// TwinCAT 3 PLC project VekSi_PLC
// ProgramVersion: 3.1.4026.22
// libraries:
//   Tc2_MC2, * (Beckhoff Automation GmbH)
//   Tc2_Standard, * (Beckhoff Automation GmbH)
//   Tc2_System, * (Beckhoff Automation GmbH)
//   Tc2_Utilities, * (Beckhoff Automation GmbH)
//   Tc3_IotBase, * (Beckhoff Automation GmbH)
//   Tc3_JsonXml, * (Beckhoff Automation GmbH)
// project tree:
//   Functions/ FB_CSVLogger.TcPOU, FB_ValveControl.TcPOU, FB_MqttManager.TcPOU, FB_SensorIO.TcPOU, MAIN.TcPOU
//   / PlcTask.TcTTO (not stored)
//   State_Var/ E_CSVLogState.TcDUT (not stored), E_MQTTState.TcDUT, E_CommandSource.TcDUT, E_ValveState.TcDUT, ST_MqttConfig.TcDUT, ST_MQTT_Command.TcDUT, ST_SensorData.TcDUT, ST_ValveData.TcDUT
//   Variables_Lists/ GVL_Config.TcGVL, GVL_HMI.TcGVL, GVL_IO.TcGVL, GVL_System.TcGVL
// real-time tasks:
//   TASK PlcTask: cycle T#10ms, priority 20, ADS port 350
// motion (NC):
//   TASK NC-Task 1 SAF: cycle T#2ms, priority 4, ADS port 501
//   TASK NC-Task 1 SVB: cycle T#10ms, priority 8, ADS port 511
//   AXIS Axis 2 (id 2)
//     Dynamic: Acceleration=16.9085, Deceleration=16.9085, Jerk=53.5391
//     Velo: RefSearch=3, RefSync=3, SlowManual=2, FastManual=3, Fast=3, Maximum=6
//     OtherSettings: AllowMotionCmdToSlave=true
//     encoder EncType=1
//       EncPara: ScaleFactorNumerator=0.003048
//         Inc: RefSoftSyncMask=#x0000ffff, HomingSensorSource=1
//         TimeComp: TimeCompMode=1, EncDelayCycles=4
//     drive DrvType=24
//       Analog: VeloReferenz=6.096, TorqueSetpointScale=10, ScaleFactorActTorque=0.1
//       TimeComp: TaskDelayCycles=1
//     controller CtrType=1
//       CtrPara: PriorControlFactor=1
//         PosDiffControl: Enable=false
//         Observer: BandWidth=20
//   AXIS Axis 3 (id 3)
//     Dynamic: Acceleration=16.9085, Deceleration=16.9085, Jerk=53.5391
//     Velo: RefSearch=3, RefSync=3, SlowManual=2, FastManual=3, Maximum=6
//     OtherSettings: AllowMotionCmdToSlave=true
//     encoder EncType=1
//       EncPara: ScaleFactorNumerator=0.003048
//         Inc: RefSoftSyncMask=#x0000ffff
//         TimeComp: TimeCompMode=1, EncDelayCycles=4
//     drive DrvType=24
//       Analog: VeloReferenz=6.096, TorqueSetpointScale=10, ScaleFactorActTorque=0.1
//       TimeComp: TaskDelayCycles=1
//     controller CtrType=1
//       CtrPara: PriorControlFactor=1
//         PosDiffControl: Enable=false
//         Observer: BandWidth=20
//   AXIS Axis 1 (id 1)
//     Dynamic: Acceleration=16.9085, Deceleration=16.9085, Jerk=53.5391
//     Velo: RefSearch=3, RefSync=3, SlowManual=2, FastManual=3, Maximum=6
//     OtherSettings: AllowMotionCmdToSlave=true
//     encoder EncType=1
//       EncPara: ScaleFactorNumerator=0.003048
//         Inc: RefSearchInverse=true, RefSyncInverse=false, RefSoftSyncMask=#x0000ffff
//         TimeComp: TimeCompMode=1, EncDelayCycles=4
//     drive DrvType=24
//       Analog: VeloReferenz=6.096, TorqueSetpointScale=10, ScaleFactorActTorque=0.1
//       TimeComp: TaskDelayCycles=1
//     controller CtrType=1
//       CtrPara: PriorControlFactor=1
//         PosDiffControl: Enable=false
//         Observer: BandWidth=20
// I/O:
//   DEVICE Device 1 (EtherCAT), AmsNetId 10.1.176.203.2.1
//     Term 1 (EK1200) [EK1200-5000 EtherCAT Power supply (2A E-Bus)]
//       Term 2 (EL6070-0033) [EL6070-0033 1Ch. Licence key terminal, individual licences]
//       Term 3 (EL1859) [EL1859 8Ch. Dig. Input 24V, 3ms, 8Ch. Dig. Output 24V, 0.5A]
//       Term 4 (EL3202) [EL3202 2Ch. Ana. Input PT100 (RTD)]
//       Term 5 (EL1004) [EL1004 4Ch. Dig. Input 24V, 3ms]
//       Term 6 (EL3074) [EL3074 4Ch. Ana. Input +/-10V, +/-20mA]
//       Term 7 (EK1322) [EK1322 2-port EtherCAT P junction with feed-in]
//         Box 8 (EPP7041-1002) [EPP7041-1002 1Ch. Stepper motor output stage (50V, 1.5A)]
//       Term 9 (EK1521-0010) [EK1521-0010 1 port EtherCAT junction (FX-SingleMode)]
//         Term 10 (EK1501-0010) [EK1501-0010 EtherCAT Coupler (2A E-Bus, FX-SingleMode, ID switch)]
//           Term 11 (EL3202) [EL3202 2Ch. Ana. Input PT100 (RTD)]
//           Term 12 (EL1859) [EL1859 8Ch. Dig. Input 24V, 3ms, 8Ch. Dig. Output 24V, 0.5A]
//           Term 13 (EL3074) [EL3074 4Ch. Ana. Input +/-10V, +/-20mA]
//           Term 22 (EL9011) [EL9011 End Terminal]
//       Term 14 (EK1521-0010) [EK1521-0010 1 port EtherCAT junction (FX-SingleMode)]
//         Term 15 (EK1501-0010) [EK1501-0010 EtherCAT Coupler (2A E-Bus, FX-SingleMode, ID switch)]
//           Term 16 (EL3202) [EL3202 2Ch. Ana. Input PT100 (RTD)]
//           Term 17 (EL1004) [EL1004 4Ch. Dig. Input 24V, 3ms]
//           Term 18 (EL3074) [EL3074 4Ch. Ana. Input +/-10V, +/-20mA]
//           Term 19 (EK1322) [EK1322 2-port EtherCAT P junction with feed-in]
//             Box 20 (EPP7041-1002) [EPP7041-1002 1Ch. Stepper motor output stage (50V, 1.5A)]
//             Box 21 (EPP7041-1002) [EPP7041-1002 1Ch. Stepper motor output stage (50V, 1.5A)]
// variable links:
//   NC-Task 1 SAF/Axes/Axis 1 <-> Device 1 (EtherCAT)/Term 1 (EK1200)/Term 7 (EK1322)/Box 8 (EPP7041-1002)
//     Drive/Inputs/In/nState1 @bit 3 <-> STM Status/Status/Error
//     Drive/Inputs/In/nState1 @bit 7 <-> STM Status/Status/Motor stall
//     Drive/Inputs/In/nState1 @bit 5 <-> STM Status/Status/Moving negative
//     Drive/Inputs/In/nState1 @bit 4 <-> STM Status/Status/Moving positive
//     Drive/Inputs/In/nState1 @bit 1 <-> STM Status/Status/Ready
//     Drive/Inputs/In/nState1 <-> STM Status/Status/Ready to enable
//     Drive/Inputs/In/nState1 @bit 6 <-> STM Status/Status/Torque reduced
//     Drive/Inputs/In/nState1 @bit 2 <-> STM Status/Status/Warning
//     Drive/Inputs/In/nState2 @bit 5 <-> STM Status/Status/Sync error
//     Drive/Inputs/In/nState2 @bit 7 <-> STM Status/Status/TxPDO Toggle
//     Drive/Inputs/In/nState4 @bit 1 <-> WcState/InputToggle
//     Drive/Inputs/In/nState4 <-> WcState/WcState
//     Drive/Outputs/Out/nCtrl1 <-> STM Control/Control/Enable
//     Drive/Outputs/Out/nCtrl1 @bit 2 <-> STM Control/Control/Reduce torque
//     Drive/Outputs/Out/nCtrl1 @bit 1 <-> STM Control/Control/Reset
//     Drive/Outputs/Out/nCtrl2 @bit 3 <-> STM Control/Control/Digital output 1
//     Drive/Outputs/Out/nDataOut2[0] <-> STM Velocity/Velocity
//   NC-Task 1 SAF/Axes/Axis 2 <-> Device 1 (EtherCAT)/Term 1 (EK1200)/Term 14 (EK1521-0010)/Term 15 (EK1501-0010)/Term 19 (EK1322)/Box 20 (EPP7041-1002)
//     Drive/Inputs/In/nState1 @bit 3 <-> STM Status/Status/Error
//     Drive/Inputs/In/nState1 @bit 7 <-> STM Status/Status/Motor stall
//     Drive/Inputs/In/nState1 @bit 5 <-> STM Status/Status/Moving negative
//     Drive/Inputs/In/nState1 @bit 4 <-> STM Status/Status/Moving positive
//     Drive/Inputs/In/nState1 @bit 1 <-> STM Status/Status/Ready
//     Drive/Inputs/In/nState1 <-> STM Status/Status/Ready to enable
//     Drive/Inputs/In/nState1 @bit 6 <-> STM Status/Status/Torque reduced
//     Drive/Inputs/In/nState1 @bit 2 <-> STM Status/Status/Warning
//     Drive/Inputs/In/nState2 @bit 3 <-> STM Status/Status/Digital input 1
//     Drive/Inputs/In/nState2 @bit 4 <-> STM Status/Status/Digital input 2
//     Drive/Inputs/In/nState2 @bit 5 <-> STM Status/Status/Sync error
//     Drive/Inputs/In/nState2 @bit 7 <-> STM Status/Status/TxPDO Toggle
//     Drive/Inputs/In/nState4 @bit 1 <-> WcState/InputToggle
//     Drive/Inputs/In/nState4 <-> WcState/WcState
//     Drive/Outputs/Out/nCtrl1 <-> STM Control/Control/Enable
//     Drive/Outputs/Out/nCtrl1 @bit 2 <-> STM Control/Control/Reduce torque
//     Drive/Outputs/Out/nCtrl1 @bit 1 <-> STM Control/Control/Reset
//     Drive/Outputs/Out/nCtrl2 @bit 3 <-> STM Control/Control/Digital output 1
//     Drive/Outputs/Out/nDataOut2[0] <-> STM Velocity/Velocity
//     Enc/Inputs/In/nDataIn1[0] <-> ENC Status compact/Counter value
//     Enc/Inputs/In/nDataIn2[0] <-> ENC Status compact/Latch value
//     Enc/Inputs/In/nState1 @bit 4 <-> ENC Status compact/Status/Counter overflow
//     Enc/Inputs/In/nState1 @bit 3 <-> ENC Status compact/Status/Counter underflow
//     Enc/Inputs/In/nState1 @bit 7 <-> ENC Status compact/Status/Extrapolation stall
//     Enc/Inputs/In/nState1 <-> ENC Status compact/Status/Latch C valid
//     Enc/Inputs/In/nState1 @bit 1 <-> ENC Status compact/Status/Latch extern valid
//     Enc/Inputs/In/nState1 @bit 2 <-> ENC Status compact/Status/Set counter done
//     Enc/Inputs/In/nState2 @bit 4 <-> ENC Status compact/Status/Status of extern latch
//     Enc/Inputs/In/nState2 <-> ENC Status compact/Status/Status of input A
//     Enc/Inputs/In/nState2 @bit 1 <-> ENC Status compact/Status/Status of input B
//     Enc/Inputs/In/nState2 @bit 2 <-> ENC Status compact/Status/Status of input C
//     Enc/Inputs/In/nState2 @bit 5 <-> ENC Status compact/Status/Sync error
//     Enc/Inputs/In/nState2 @bit 7 <-> ENC Status compact/Status/TxPDO Toggle
//     Enc/Inputs/In/nState4 @bit 1 <-> WcState/InputToggle
//     Enc/Inputs/In/nState4 <-> WcState/WcState
//     Enc/Outputs/Out/nCtrl1 <-> ENC Control compact/Control/Enable latch C
//     Enc/Outputs/Out/nCtrl1 @bit 3 <-> ENC Control compact/Control/Enable latch extern on negative edge
//     Enc/Outputs/Out/nCtrl1 @bit 1 <-> ENC Control compact/Control/Enable latch extern on positive edge
//     Enc/Outputs/Out/nCtrl1 @bit 2 <-> ENC Control compact/Control/Set counter
//     Enc/Outputs/Out/nDataOut1[0] <-> ENC Control compact/Set counter value
//   NC-Task 1 SAF/Axes/Axis 3 <-> Device 1 (EtherCAT)/Term 1 (EK1200)/Term 14 (EK1521-0010)/Term 15 (EK1501-0010)/Term 19 (EK1322)/Box 21 (EPP7041-1002)
//     Drive/Inputs/In/nState1 @bit 3 <-> STM Status/Status/Error
//     Drive/Inputs/In/nState1 @bit 7 <-> STM Status/Status/Motor stall
//     Drive/Inputs/In/nState1 @bit 5 <-> STM Status/Status/Moving negative
//     Drive/Inputs/In/nState1 @bit 4 <-> STM Status/Status/Moving positive
//     Drive/Inputs/In/nState1 @bit 1 <-> STM Status/Status/Ready
//     Drive/Inputs/In/nState1 <-> STM Status/Status/Ready to enable
//     Drive/Inputs/In/nState1 @bit 6 <-> STM Status/Status/Torque reduced
//     Drive/Inputs/In/nState1 @bit 2 <-> STM Status/Status/Warning
//     Drive/Inputs/In/nState2 @bit 3 <-> STM Status/Status/Digital input 1
//     Drive/Inputs/In/nState2 @bit 4 <-> STM Status/Status/Digital input 2
//     Drive/Inputs/In/nState2 @bit 5 <-> STM Status/Status/Sync error
//     Drive/Inputs/In/nState2 @bit 7 <-> STM Status/Status/TxPDO Toggle
//     Drive/Inputs/In/nState4 @bit 1 <-> WcState/InputToggle
//     Drive/Inputs/In/nState4 <-> WcState/WcState
//     Drive/Outputs/Out/nCtrl1 <-> STM Control/Control/Enable
//     Drive/Outputs/Out/nCtrl1 @bit 2 <-> STM Control/Control/Reduce torque
//     Drive/Outputs/Out/nCtrl1 @bit 1 <-> STM Control/Control/Reset
//     Drive/Outputs/Out/nCtrl2 @bit 3 <-> STM Control/Control/Digital output 1
//     Drive/Outputs/Out/nDataOut2[0] <-> STM Velocity/Velocity
//     Enc/Inputs/In/nDataIn1[0] <-> ENC Status compact/Counter value
//     Enc/Inputs/In/nDataIn2[0] <-> ENC Status compact/Latch value
//     Enc/Inputs/In/nState1 @bit 4 <-> ENC Status compact/Status/Counter overflow
//     Enc/Inputs/In/nState1 @bit 3 <-> ENC Status compact/Status/Counter underflow
//     Enc/Inputs/In/nState1 @bit 7 <-> ENC Status compact/Status/Extrapolation stall
//     Enc/Inputs/In/nState1 <-> ENC Status compact/Status/Latch C valid
//     Enc/Inputs/In/nState1 @bit 1 <-> ENC Status compact/Status/Latch extern valid
//     Enc/Inputs/In/nState1 @bit 2 <-> ENC Status compact/Status/Set counter done
//     Enc/Inputs/In/nState2 @bit 4 <-> ENC Status compact/Status/Status of extern latch
//     Enc/Inputs/In/nState2 <-> ENC Status compact/Status/Status of input A
//     Enc/Inputs/In/nState2 @bit 1 <-> ENC Status compact/Status/Status of input B
//     Enc/Inputs/In/nState2 @bit 2 <-> ENC Status compact/Status/Status of input C
//     Enc/Inputs/In/nState2 @bit 5 <-> ENC Status compact/Status/Sync error
//     Enc/Inputs/In/nState2 @bit 7 <-> ENC Status compact/Status/TxPDO Toggle
//     Enc/Inputs/In/nState4 @bit 1 <-> WcState/InputToggle
//     Enc/Inputs/In/nState4 <-> WcState/WcState
//     Enc/Outputs/Out/nCtrl1 <-> ENC Control compact/Control/Enable latch C
//     Enc/Outputs/Out/nCtrl1 @bit 3 <-> ENC Control compact/Control/Enable latch extern on negative edge
//     Enc/Outputs/Out/nCtrl1 @bit 1 <-> ENC Control compact/Control/Enable latch extern on positive edge
//     Enc/Outputs/Out/nCtrl1 @bit 2 <-> ENC Control compact/Control/Set counter
//     Enc/Outputs/Out/nDataOut1[0] <-> ENC Control compact/Set counter value
//   VekSi_PLC/VekSi_PLC Instance <-> Device 1 (EtherCAT)/Term 1 (EK1200)/Term 7 (EK1322)/Box 8 (EPP7041-1002)
//     PlcTask Inputs/GVL_IO.bBottom_position_1 <-> STM Status/Status/Digital input 1
//     PlcTask Inputs/GVL_IO.bTop_position_1 <-> STM Status/Status/Digital input 2
//   VekSi_PLC/VekSi_PLC Instance <-> NC-Task 1 SAF/Axes/Axis 1
//     PlcTask Inputs/MAIN.Axis_Valve1.NcToPlc <-> Outputs/ToPlc
//     PlcTask Outputs/MAIN.Axis_Valve1.PlcToNc <-> Inputs/FromPlc
//   VekSi_PLC/VekSi_PLC Instance <-> NC-Task 1 SAF/Axes/Axis 2
//     PlcTask Inputs/MAIN.Axis_Valve2.NcToPlc <-> Outputs/ToPlc
//     PlcTask Outputs/MAIN.Axis_Valve2.PlcToNc <-> Inputs/FromPlc
//   VekSi_PLC/VekSi_PLC Instance <-> NC-Task 1 SAF/Axes/Axis 3
//     PlcTask Inputs/MAIN.Axis_Valve3.NcToPlc <-> Outputs/ToPlc
//     PlcTask Outputs/MAIN.Axis_Valve3.PlcToNc <-> Inputs/FromPlc

// ---- State_Var/E_MQTTState.TcDUT
{attribute 'qualified_only'}
{attribute 'strict'}
{attribute 'to_string'}
TYPE E_MQTTState :
(
	DISABLED := 0,
    CONNECTING := 1,
    CONNECTED := 2,
    DISCONNECTING := 3,
    WAIT_RECONNECT := 4
);
END_TYPE

// ---- State_Var/E_CommandSource.TcDUT
{attribute 'qualified_only'}
{attribute 'strict'}
{attribute 'to_string'}
TYPE E_CommandSource :
(
    HMI    := 0,   // Commands are taken from the local HMI
    MQTT   := 1,   // Commands are taken from MQTT when enabled and connected
    Manual := 2    // Commands are taken from future local/manual inputs
);
END_TYPE

// ---- State_Var/E_ValveState.TcDUT
{attribute 'qualified_only'}
{attribute 'strict'}
{attribute 'to_string'}
TYPE E_ValveState :
(
    INIT    		:= 0,   // Initializing, powering axis
    HOMING  		:= 1,   // Performing homing sequence (MC_Home)
    IDLE    		:= 2,   // At position, no active command
    MOVING  		:= 3,   // MC_MoveAbsolute active, travelling to setpoint
	HALT			:= 4,
    HOLD		    := 5,   // At setpoint, holding position
    MANNUAL_JOG		:= 6, // Manual hardware-panel jog mode
    FAULT   		:= 7,   // Error state — MC error, drive fault, or limit breach
    RESET   		:= 8    // Clearing fault, preparing to re-home
);
END_TYPE

// ---- State_Var/ST_MqttConfig.TcDUT
(*
============================================================
ST_MqttConfig
============================================================
PURPOSE
  MQTT broker connection and topic configuration.
  Populated from GVL_Config defaults on startup.
  Operator can override all fields from the HMI MQTT-Config
  panel, then press "Apply & Reconnect" to activate changes.

NOTES
  • Changing any field requires pressing Apply (triggers bApplyConfig
    rising edge in FB_MqttManager) to reconnect with new settings.
  • Use TLS (bUseTls = TRUE, nPort = 8883) for production deployments.
  • Credentials are NOT stored in persistent memory — they must be
    re-entered after a cold restart unless the HMI retains them.
============================================================
*)
TYPE ST_MqttConfig :
STRUCT
    (* ── Broker Connection ──────────────────────────────────── *)
    sBrokerAddress      : STRING(255) := 'imsiot.aws.thinger.io';   (* IP or hostname of MQTT broker     *)
    nPort               : UINT        := 1883;              (* 1883 = plain, 8883 = TLS/SSL      *)
    sClientId           : STRING(64)  := 'Beckhoff'; (* Must be unique per broker   *)
    sUsername           : STRING(64)  := 'ims_iot';                (* Leave empty if no auth required   *)
    sPassword           : STRING(64)  := '123456789';                (* Leave empty if no auth required   *)
    bUseTls             : BOOL        := FALSE;             (* TRUE enables TLS/SSL connection   *)

    (* ── Topic Configuration ────────────────────────────────── *)
    sTopicPrefix        : STRING(64)  := 'irrigation';      (* Base prefix for all topics        *)
    (* Publish topic  : <prefix>/status                                                           *)
    (* Subscribe topic: <prefix>/command                                                          *)
    sMainTopic          : STRING(128) := 'irrigation/status';   (* Full publish topic            *)
    SubscribeTopic      : STRING(128) := 'irrigation/command';  (* Full subscribe topic          *)

    (* ── Timing ─────────────────────────────────────────────── *)
    tStatusPublishInterval : TIME := T#5M;                  (* Cyclic publish interval (5 min)   *)
    tReconnectDelay        : TIME := T#30S;                 (* Back-off delay between retries    *)

    (* ── Runtime Control ────────────────────────────────────── *)
    bUseStatusPublish   : BOOL := TRUE;                     (* TRUE = publish status cyclically  *)
    bApplyConfig        : BOOL;                             (* Rising edge: reconnect with new cfg*)
END_STRUCT
END_TYPE

// ---- State_Var/ST_MQTT_Command.TcDUT
(*
============================================================
ST_MQTT_Command
============================================================
PURPOSE
  JSON-deserialized incoming MQTT command payload.
  FB_MqttManager parses received JSON into this struct.

EXPECTED JSON FORMAT (publish to irrigation/command):
  {
    "Valve1": 50,
    "Valve2": 25,
    "Valve3": 75
  }

  Valve setpoints are in percent (0–100).
  Omitting a field leaves its current value unchanged.

NOTES
  • {attribute 'TcJsonObject'} enables Beckhoff JSON auto-parse.
  • DINT used for setpoints to avoid floating-point JSON quirks;
    values are clamped to 0–100 before use.
============================================================
*)
{attribute 'TcJsonObject' := ''}
TYPE ST_MQTT_Command :
STRUCT
    (* ── Setpoints (0–100 %) ────────────────────────────────── *)
    Valve1          : DINT;     (* Desired position valve 1, 0–100 % *)
    Valve2          : DINT;     (* Desired position valve 2, 0–100 % *)
    Valve3          : DINT;     (* Desired position valve 3, 0–100 % *)
END_STRUCT
END_TYPE

// ---- State_Var/ST_SensorData.TcDUT
(*
============================================================
ST_SensorData
============================================================
PURPOSE
  Holds all sensor readings converted to engineering units.
  Populated by FB_SensorIO every PLC cycle.
  Consumed by MAIN, FB_CSVLogger, and FB_MqttManager.

WATER LEVEL
  Three sensors: L1V11 (primary), L1V20 (secondary), L2V21 (tertiary).
  rWaterLevel_pct  — percentage 0–100 % (primary sensor only).
  rWaterLevel_mm   — absolute level in mm (primary sensor only).

TEMPERATURE
  Two channels from EL3202 RTD card.
  rTemperature_C[1] — Probe 1 in degrees Celsius.
  rTemperature_C[2] — Probe 2 in degrees Celsius.

POSITION FEEDBACK (encoder)
  Raw encoder counts scaled to mm for each valve axis.
  rPosFeedback_mm[1..3] — supplementary position, not used by MC2
  (MC2 reads encoder directly via NC axis).

FAULT FLAGS
  bWaterLevelFault — raw value below disconnection threshold.
  bTempFault[1..2] — raw value below disconnection threshold.
============================================================
*)
TYPE ST_SensorData :
STRUCT
    (* ── Water Level ────────────────────────────────────────── *)
    rWaterLevel_pct         : REAL;             (* Primary sensor: 0–100 %           *)
    rWaterLevel_mm          : REAL;             (* Primary sensor: 0–ENG_MAX mm      *)
    rWaterLevel_raw         : INT;              (* Raw ADC value for diagnostics      *)
    bWaterLevelFault        : BOOL;             (* TRUE if sensor disconnected/out-rng*)

    (* ── Temperature ────────────────────────────────────────── *)
    rTemperature_C          : ARRAY[1..2] OF REAL;  (* Probe 1 and 2 in °C           *)
    rTemperature_raw        : ARRAY[1..2] OF INT;   (* Raw ADC values for diagnostics *)
    bTempFault              : ARRAY[1..2] OF BOOL;  (* TRUE if sensor fault           *)

    (* ── Position Feedback (supplementary, NC reads directly) ─ *)
    rPosFeedback_mm         : ARRAY[1..3] OF REAL;  (* Encoder position in mm         *)
    rPosFeedback_raw        : ARRAY[1..3] OF INT;   (* Raw counts for diagnostics     *)
    bPosFeedbackFault       : ARRAY[1..3] OF BOOL;  (* TRUE if encoder disconnected   *)

    (* ── Aggregate Health ───────────────────────────────────── *)
    bAnySensorFault         : BOOL;             (* OR of all fault flags              *)
END_STRUCT
END_TYPE

// ---- State_Var/ST_ValveData.TcDUT

TYPE ST_ValveData :
STRUCT
    // --- Setpoints (written by HMI or MQTT) ---
    HMI_Setpoint    : REAL;         // Position setpoint from HMI (0.0–100.0 %)
    MQTT_Setpoint   : REAL;         // Position setpoint from MQTT (0.0–100.0 %)
    Manual_Setpoint : REAL;         // Future local/manual position setpoint (0.0–100.0 %)
    Active_Setpoint : REAL;         // Currently selected setpoint after source arbitration

    // --- Feedback (written by FB_ValveControl) ---
    Actual_Position : REAL;         // Actual valve position in % (from MC axis)
    Actual_Pos_Raw  : LREAL;        // Raw axis position in mm or steps (from MC2)

    // --- Command source tracking ---
    Source          : E_CommandSource;  
	lastsrc			: E_CommandSource; // Who issued the last command
	

    // --- State machine status ---
    State           	: E_ValveState;  // Current state of FB_ValveControl
	currentState_string : STRING;
    IsHomed         	: BOOL;          // TRUE once homing has been completed
    InPosition      	: BOOL;          // TRUE when actual ≈ setpoint (within tolerance)
    IsFault         	: BOOL;          // TRUE when in FAULT state
    FaultCode       	: UDINT;         // MC or drive error code for diagnostics
	

	
    // --- Reset ---
    Reset_Cmd       : BOOL;          // HMI writes TRUE to request fault reset
END_STRUCT
END_TYPE

// ---- Variables_Lists/GVL_Config.TcGVL
(*
============================================================
GVL_Config  —  System-wide compile-time constants
============================================================
All values here are CONSTANT and cannot be changed at runtime.
To change a value: edit here, rebuild and download the project.
Runtime-adjustable parameters are exposed via GVL_HMI.

CALIBRATION REQUIRED:
  • VALVE_FULL_STROKE_MM  — measure physical travel of each actuator
  • WATER_LEVEL_ENG_MAX_MM — measure the full-scale tank height
  • Sensor raw min/max    — verify with your specific EL3074 settings
============================================================
*)
{attribute 'qualified_only'}
VAR_GLOBAL CONSTANT

    // ── Valve Motion Parameters ─────────────────────────────────
    // *** CALIBRATE to hardware before first run ***
    VALVE_FULL_STROKE_MM        : REAL   := 126;      // mm — full travel (3600° stepper)
    VALVE_POSITION_TOLERANCE    : REAL   := 0.5;        // %  — in-position dead-band
    VALVE_MOVE_VELOCITY         : LREAL  := 1.5;        // mm/s — max travel speed
    VALVE_MOVE_ACCELERATION     : LREAL  := 16.9085;    // mm/s² — ramp-up rate
    VALVE_MOVE_DECELERATION     : LREAL  := 16.9085;    // mm/s² — ramp-down rate
    VALVE_MOVE_JERK             : LREAL  := 53.5391;    // mm/s³ — 0.0 = trapezoidal profile
    VALVE_HOMING_VELOCITY       : LREAL  := 1.0;        // mm/s — slow speed during homing

    // ── Sensor Scaling — Water Level ───────────────────────────
    // Raw INT from EL3074 (4–20 mA, 0–32767 counts typical)
    // Adjust RAW_MIN/MAX to match your EL3074 configuration
    WATER_LEVEL_RAW_MIN         : INT    := 0;          // ADC count at 0 % / 0 mm
    WATER_LEVEL_RAW_MAX         : INT    := 32767;      // ADC count at 100 % / ENG_MAX_MM
    WATER_LEVEL_ENG_MIN_MM      : REAL   := 0.0;        // mm at raw minimum
    WATER_LEVEL_ENG_MAX_MM      : REAL   := 1000.0;     // mm at raw maximum — calibrate!

    // ── Sensor Scaling — Temperature ───────────────────────────
    // Raw INT from EL3202 RTD (PT100, -200…+850 °C, 0.1 °C resolution)
    // EL3202 outputs tenths of a degree, e.g. 250 = 25.0 °C
    TEMP_RAW_SCALE_FACTOR       : REAL   := 0.1;        // °C per raw count
    TEMP_OFFSET_C               : REAL   := 0.0;        // offset correction if needed

    // ── Sensor Fault Detection ─────────────────────────────────
    // Readings at or below this value are treated as disconnected
    SENSOR_FAULT_THRESHOLD      : INT    := -100;       // -999 default in GVL_IO = hardware stub

    // ── CSV Logging ─────────────────────────────────────────────
    CSV_LOG_INTERVAL_S          : TIME   := T#15M;      // Logging period (15 min default)
    CSV_FILE_PATH               : STRING := 'C:\TwinCAT\3.1\Boot\Log\';
    CSV_FILENAME_PREFIX         : STRING := 'IrrigationLog_';

    // ── MQTT Defaults (loaded into GVL_HMI.HMI_MQTT_Config at startup) ──
    MQTT_DEFAULT_BROKER_IP      : STRING := 'imsiot.aws.thinger.io';
    MQTT_DEFAULT_PORT           : UINT   := 8883;
    MQTT_DEFAULT_CLIENT_ID      : STRING := 'Beckhoff';
    MQTT_DEFAULT_USERNAME       : STRING := 'ims_iot';         // Set from HMI for production
    MQTT_DEFAULT_PASSWORD       : STRING := '123456789';         // Set from HMI for production
    MQTT_DEFAULT_TOPIC_PREFIX   : STRING := 'irrigation';
    MQTT_DEFAULT_MAIN_TOPIC     : STRING := 'irrigation/status';
    MQTT_DEFAULT_SUB_TOPIC      : STRING := 'irrigation/command';
    MQTT_DEFAULT_PUBLISH_INTERVAL : UINT := 300;        // 300 s = 5 min

    // ── Task Cycle Time ──────────────────────────────────────────
    TASK_CYCLE_MS               : UINT   := 10;         // Must match TwinCAT task setting

END_VAR

// ---- Variables_Lists/GVL_HMI.TcGVL
(*
============================================================
GVL_HMI  —  HMI ↔ PLC interface layer
============================================================
PURPOSE
  All variables in this GVL are bound to TcHMI controls via
  the ADS symbol server. HMI_* variables are written by the
  operator (HMI inputs). ACT_* variables are written by the
  PLC (HMI outputs / displays).

NAMING CONVENTION
  HMI_*   → HMI writes, PLC reads  (operator commands)
  ACT_*   → PLC writes, HMI reads  (status displays)

BINDING PATTERN (TcHMI)
  %s%ADS.PLC1.GVL_HMI.<VariableName>%/s%
============================================================
*)
VAR_GLOBAL

    // ══════════════════════════════════════════════════════════
    // COMMAND SOURCE SELECTION
    // ══════════════════════════════════════════════════════════
    HMI_CommandSource           : E_CommandSource := E_CommandSource.HMI; // HMI input: selected command source for all valves

    // ══════════════════════════════════════════════════════════
    // VALVE 1 — HMI Interface
    // ══════════════════════════════════════════════════════════
    HMI_Valve1_Setpoint         : REAL;             // HMI input:  desired position 0–100 %
    HMI_Valve1_Reset            : BOOL;             // HMI button: reset fault for valve 1
    HMI_Valve1_Stop             : BOOL;             // HMI button: halt valve 1 movement
    HMI_Valve1_Homing           : BOOL;             // HMI button: trigger re-homing valve 1
    HMI_UPDATE                  : BOOL;             // HMI button: apply setpoint(s)

    ACT_Valve1_Position         : REAL;             // PLC output: actual position 0–100 %
    ACT_Valve1_State            : STRING;     // PLC output: current state machine state
    ACT_Valve1_Source           : E_CommandSource;    // PLC output: last command source enum
    ACT_Valve1_SourceText       : STRING(8);        // PLC output: 'HMI', 'MQTT', 'Manual', or 'NONE'
    ACT_Valve1_Fault            : BOOL;             // PLC output: fault active flag
    ACT_Valve1_FaultCode        : UDINT;            // PLC output: MC2 fault code
    Raw_Valve1_Setpoint         : LREAL;            // PLC output: active setpoint in mm
    Raw_Valve1_Position         : LREAL;            // PLC output: actual position in mm
	

    // ══════════════════════════════════════════════════════════
    // VALVE 2 — HMI Interface
    // ══════════════════════════════════════════════════════════
    HMI_Valve2_Setpoint         : REAL;             // HMI input:  desired position 0–100 %
    HMI_Valve2_Reset            : BOOL;             // HMI button: reset fault for valve 2
    HMI_Valve2_Stop             : BOOL;             // HMI button: halt valve 2 movement
    HMI_Valve2_Homing           : BOOL;             // HMI button: trigger re-homing valve 2

    ACT_Valve2_Position         : REAL;             // PLC output: actual position 0–100 %
    ACT_Valve2_State            : STRING;     // PLC output: current state machine state
    ACT_Valve2_Source           : E_CommandSource;    // PLC output: last command source enum
    ACT_Valve2_SourceText       : STRING(8);        // PLC output: 'HMI', 'MQTT', 'Manual', or 'NONE'
    ACT_Valve2_Fault            : BOOL;             // PLC output: fault active flag
    ACT_Valve2_FaultCode        : UDINT;            // PLC output: MC2 fault code
    Raw_Valve2_Setpoint         : LREAL;            // PLC output: active setpoint in mm
    Raw_Valve2_Position         : LREAL;            // PLC output: actual position in mm

    // ══════════════════════════════════════════════════════════
    // VALVE 3 — HMI Interface
    // ══════════════════════════════════════════════════════════
    HMI_Valve3_Setpoint         : REAL;             // HMI input:  desired position 0–100 %
    HMI_Valve3_Reset            : BOOL;             // HMI button: reset fault for valve 3
    HMI_Valve3_Stop             : BOOL;             // HMI button: halt valve 3 movement
    HMI_Valve3_Homing           : BOOL;             // HMI button: trigger re-homing valve 3

    ACT_Valve3_Position         : REAL;             // PLC output: actual position 0–100 %
    ACT_Valve3_State            : STRING;     // PLC output: current state machine state
    ACT_Valve3_Source           : E_CommandSource;    // PLC output: last command source enum
    ACT_Valve3_SourceText       : STRING(8);        // PLC output: 'HMI', 'MQTT', 'Manual', or 'NONE'
    ACT_Valve3_Fault            : BOOL;             // PLC output: fault active flag
    ACT_Valve3_FaultCode        : UDINT;            // PLC output: MC2 fault code
    Raw_Valve3_Setpoint         : LREAL;            // PLC output: active setpoint in mm
    Raw_Valve3_Position         : LREAL;            // PLC output: actual position in mm

    // ══════════════════════════════════════════════════════════
    // SENSOR DISPLAYS
    // ══════════════════════════════════════════════════════════
    ACT_WaterLevel_pct          : REAL;             // PLC output: water level 0–100 %
    ACT_WaterLevel_mm           : REAL;             // PLC output: water level in mm
    ACT_Temperature1_C          : REAL;             // PLC output: temperature probe 1 (°C)
    ACT_Temperature2_C          : REAL;             // PLC output: temperature probe 2 (°C)
    ACT_SensorFault             : BOOL;             // PLC output: any sensor disconnected

    // ══════════════════════════════════════════════════════════
    // MQTT CONTROL & STATUS
    // ══════════════════════════════════════════════════════════
    HMI_MQTT_bEnable            : BOOL;             // HMI checkbox: system MQTT connection enable
    HMI_MQTT_mPublish           : BOOL;             // HMI button:   manual publish now
    HMI_MQTT_Config             : ST_MqttConfig;    // HMI panel:    broker configuration
    HMI_MQTT_ApplyConfig        : BOOL;             // HMI button:   apply config & reconnect

    ACT_MQTT_Connected          : BOOL;             // PLC output: broker connection active
	ACT_MQTT_State				: STRING;
    ACT_MQTT_Error              : BOOL;             // PLC output: connection error flag
    ACT_MQTT_ErrorMsg           : STRING(128);      // PLC output: error description text
    ACT_MQTT_JsonPreview        : STRING(2048);     // PLC output: last outgoing JSON (debug)
    ACT_MQTT_LastMsgRcvTime		: STRING;
	ACT_MQTT_LastMsgPubTime		: STRING;
	ACT_MQTT_LastRxTopic        : STRING(255);      // PLC output: last received topic
    ACT_MQTT_NewCommand         : BOOL;             // PLC output: TRUE for one cycle on cmd
	

    // ══════════════════════════════════════════════════════════
    // CSV LOGGER CONTROL & STATUS
    // ══════════════════════════════════════════════════════════
    HMI_CSV_Enable              : BOOL := TRUE;     // HMI checkbox: enable logging
    WriteTrigger                : BOOL;             // HMI button:   force write a row now
    ACT_CSV_CurrentFile         : STRING;           // PLC output: active CSV filename
    ACT_CSV_LastWriteTime       : DT;               // PLC output: timestamp of last write
    ACT_CSV_Error               : BOOL;             // PLC output: file I/O error

    // ══════════════════════════════════════════════════════════
    // SYSTEM-WIDE CONTROLS & STATUS
    // ══════════════════════════════════════════════════════════
    HMI_ResetAll                : BOOL;             // HMI button: reset all valve faults
    ACT_SystemReady             : BOOL;             // PLC output: all homed, no faults
	
	
	///////HMI Control signals
	
	sHMI_mode		: BOOL;
	sMqtt_mode		: BOOL;
	sMannual_mode	: BOOL;
	
	
	
	
	

END_VAR

// ---- Variables_Lists/GVL_IO.TcGVL
{attribute 'qualified_only'}
VAR_GLOBAL
	
	AI_L1V11  					: INT	:= -999 ;	// AT %I* // Water Level Sensors
	AI_L1V20  					: INT	:= -999 ;	// AT %I*
	AI_L2V21  					: INT	:= -999 ;	// AT %I*

	AI_Tmp_1 					: INT	:= -999;	// AT %I*
	AI_Tmp_2  					: INT	:= -999;	// AT %I*
	
	AI_PosFeedback_1			: INT	:= -999;	// AT %I* //Position feedback from the encoder
	AI_PosFeedback_2			: INT	:= -999;	// AT %I*
	AI_PosFeedback_3			: INT	:= -999;	// AT %I*

	bTop_position_1		AT %I*	: BOOL;
	bBottom_position_1	AT %I*	: BOOL;
	
	///////need to add links later/////////////////
	
	bTop_position_2			: BOOL;
	bBottom_position_2		: BOOL;
	
  	bTop_position_3			: BOOL;
	bBottom_position_3		: BOOL;
	// Local panel jog push buttons (physical inputs)
	bValve1_JogUp_PB		: BOOL;
	bValve1_JogDown_PB		: BOOL;
	
	bValve2_JogUp_PB		: BOOL;
	bValve2_JogDown_PB		: BOOL;
	
	bValve3_JogUp_PB		: BOOL;
	bValve3_JogDown_PB		: BOOL;
	// Local panel jog indicator LEDs (physical outputs)
	bValve1_JogUp_LED		: BOOL;
	bValve1_JogDown_LED		: BOOL;
	
	bValve2_JogUp_LED		: BOOL;
	bValve2_JogDown_LED		: BOOL;
	
	bValve3_JogUp_LED		: BOOL;
	bValve3_JogDown_LED		: BOOL;
	
END_VAR

// ---- Variables_Lists/GVL_System.TcGVL
(*
============================================================
GVL_System  —  Runtime shared state
============================================================
PURPOSE
  Central runtime data bus. Written by function blocks,
  read by MAIN and mirrored to GVL_HMI for display.

OWNERSHIP
  Valve[1..3]     → written by FB_ValveControl instances
  Sensors         → written by FB_SensorIO
  CSV_*           → written by FB_CSVLogger
  MQTT_*          → written by FB_MqttManager
  SystemReady,
  AnyFaultActive  → computed in MAIN
============================================================
*)
VAR_GLOBAL

    // ── Valve runtime data ───────────────────────────────────────
    Valve                   : ARRAY[1..3] OF ST_ValveData;  // Index 1=V1, 2=V2, 3=V3
	bCommandUpdate_MQTT			: BOOL;
	bCommandUpdate_HMI			: BOOL;
	bCommandUpdate_Mannual		: BOOL;

	bCommandUpdate			: BOOL;

    // ── Sensor data (written by FB_SensorIO) ─────────────────────
    Sensors                 : ST_SensorData;

    // ── CSV Logger status (written by FB_CSVLogger) ───────────────
    CSV_LastWriteTime       : DT;               // Timestamp of last successful row write
    CSV_FileError           : BOOL;             // File I/O error flag
    CSV_RowsWritten         : UDINT;            // Total rows written this session
    CSV_CurrentFile         : STRING;           // Active filename (e.g. IrrigationLog_2026-04.csv)
    CSV_LoggerState         : E_CSVLogState;    // Internal state for diagnostics

    // ── MQTT runtime status (written by FB_MqttManager) ──────────
    MQTT_Connected          : BOOL;             // TRUE when broker connection is active
    MQTT_Error              : BOOL;             // TRUE on connection error or reconnect
    MQTT_LastErrorCode      : HRESULT;          // HRESULT error code (0 = OK)
    MQTT_LastErrorMsg       : STRING(128);      // Human-readable error description
    MQTT_LastRxTopic        : STRING(255);      // Last received topic
    MQTT_LastRxPayload      : STRING(2048);     // Last received payload (for diagnostics)
    MQTT_LastJsonStatus     : STRING(2048);     // Last outgoing JSON payload (for diagnostics)
    MQTT_NewCommand         : BOOL;             // TRUE for one cycle after valid command received

    // ── System health (computed in MAIN) ─────────────────────────
    SystemReady             : BOOL;             // All valves homed and no active faults
    AnyFaultActive          : BOOL;             // OR of all valve IsFault flags
    AnySensorFault          : BOOL;             // TRUE if any sensor is disconnected/faulty

END_VAR

// ---- Functions/MAIN.TcPOU
(*
============================================================
PROGRAM: MAIN
============================================================

PURPOSE
  Top-level program that orchestrates all function blocks
  and manages the system data bus between GVLs.

EXECUTION ORDER (every PLC cycle)
  1. Initialise MQTT config from defaults (first scan only)
  2. Copy HMI inputs to GVL_System bus
  3. FB_SensorIO      — Read and scale analog sensor inputs
  4. FB_ValveControl  — Per-valve TC2_MC2 state machines (x3)
  5. Build timestamp string for MQTT and logging
  6. FB_MqttManager   — MQTT connection, publish, subscribe
  7. FB_CsvLogger     — Periodic CSV row logging
  8. Mirror runtime data to GVL_HMI for display
  9. Compute system health flags

DATA FLOW
  GVL_IO  --> FB_SensorIO --> GVL_System.Sensors
  GVL_HMI.HMI_* --> GVL_System.Valve[n] setpoints
  FB_MqttManager.rMqttValveSetpoint --> FB_ValveControl MQTT_Setpoint
  FB_ValveControl outputs --> GVL_System.Valve[n] status
  GVL_System.* --> GVL_HMI.ACT_* (for display)
  GVL_System.Valve + Sensors --> FB_MqttManager (outgoing JSON)
  GVL_System.Valve + Sensors --> FB_CsvLogger (CSV row)

LIBRARIES
  TC2_MC2, TF6701 / Tc3_IotBase, Tc2_System
============================================================
*)

PROGRAM MAIN
VAR
    // ── Function block instances ────────────────────────────────
    fbSensorIO      : FB_SensorIO;    //////Not Implemented currently
    fbValve1        : FB_ValveControl;
    fbValve2        : FB_ValveControl;
    fbValve3        : FB_ValveControl;
    fbCsvLogger     : FB_CsvLogger;
    fbMqttManager   : FB_MqttManager;

    // ── NC Axis references ──────────────────────────────────────
    // Each must be linked to an NC axis in TwinCAT I/O mapping.
    Axis_Valve1     : AXIS_REF;
    Axis_Valve2     : AXIS_REF;
    Axis_Valve3     : AXIS_REF;

    // ── Timestamp for MQTT JSON ──────────────────────────────────
    fbSysTime       : FB_LocalSystemTime;
    sTimestamp      : STRING(64);
    sTempStr        : STRING(8);

    // ── Whole-array buffers passed to FB_MqttManager ─────────────
    // TwinCAT does not allow per-element array assignment inside
    // an FB call's parameter list. Populate these arrays each
    // cycle, then pass them in a single assignment.
    aValveSetpoint  : ARRAY[1..3] OF REAL;
    aValveActual    : ARRAY[1..3] OF REAL;
    aValveSource    : ARRAY[1..3] OF STRING(8);

    // ── First-scan flag for MQTT default config load ─────────────
    bMqttConfigInit : BOOL := FALSE;
	
	    // ── Local panel jog LED helpers ───────────────────────────
    bManualMode            : BOOL;

	
	rtHmiMode      : R_TRIG;
	
END_VAR

// ============================================================
// STEP 0 — ONE-TIME INITIALISATION
// On first scan, copy MQTT defaults from GVL_Config into the
// HMI-bound config struct. The operator can then edit any field
// from the HMI MQTT panel and click Apply to reconnect.
// ============================================================
IF NOT bMqttConfigInit THEN
    GVL_HMI.HMI_MQTT_Config.sBrokerAddress         := GVL_Config.MQTT_DEFAULT_BROKER_IP;
    GVL_HMI.HMI_MQTT_Config.nPort                  := GVL_Config.MQTT_DEFAULT_PORT;
    GVL_HMI.HMI_MQTT_Config.sClientId              := GVL_Config.MQTT_DEFAULT_CLIENT_ID;
    GVL_HMI.HMI_MQTT_Config.sUsername              := GVL_Config.MQTT_DEFAULT_USERNAME;
    GVL_HMI.HMI_MQTT_Config.sPassword              := GVL_Config.MQTT_DEFAULT_PASSWORD;
    GVL_HMI.HMI_MQTT_Config.sTopicPrefix           := GVL_Config.MQTT_DEFAULT_TOPIC_PREFIX;
    GVL_HMI.HMI_MQTT_Config.sMainTopic             := GVL_Config.MQTT_DEFAULT_MAIN_TOPIC;
    GVL_HMI.HMI_MQTT_Config.SubscribeTopic         := GVL_Config.MQTT_DEFAULT_SUB_TOPIC;
    GVL_HMI.HMI_MQTT_Config.tStatusPublishInterval := UDINT_TO_TIME(UINT_TO_UDINT(GVL_Config.MQTT_DEFAULT_PUBLISH_INTERVAL) * 1000);
    GVL_HMI.HMI_MQTT_Config.bUseStatusPublish      := TRUE;
   // bMqttConfigInit := TRUE;
END_IF

rtHmiMode(CLK := GVL_HMI.HMI_CommandSource = E_CommandSource.HMI);

IF rtHmiMode.Q THEN
    GVL_HMI.HMI_Valve1_Setpoint := fbValve1.Actual_Position;
    GVL_HMI.HMI_Valve2_Setpoint := fbValve2.Actual_Position;
    GVL_HMI.HMI_Valve3_Setpoint := fbValve3.Actual_Position;
END_IF

// ============================================================
// STEP 1 — COPY HMI SETPOINTS / RESETS INTO SYSTEM BUS
// ============================================================
GVL_System.Valve[1].HMI_Setpoint := GVL_HMI.HMI_Valve1_Setpoint;
GVL_System.Valve[1].Reset_Cmd    := GVL_HMI.HMI_Valve1_Reset;

GVL_System.Valve[2].HMI_Setpoint := GVL_HMI.HMI_Valve2_Setpoint;
GVL_System.Valve[2].Reset_Cmd    := GVL_HMI.HMI_Valve2_Reset;

GVL_System.Valve[3].HMI_Setpoint := GVL_HMI.HMI_Valve3_Setpoint;
GVL_System.Valve[3].Reset_Cmd    := GVL_HMI.HMI_Valve3_Reset;

GVL_System.bCommandUpdate_HMI := GVL_HMI.HMI_UPDATE; 

// Reset-All button: propagate to all valves and self-clear
IF GVL_HMI.HMI_ResetAll THEN
    GVL_System.Valve[1].Reset_Cmd := TRUE;
    GVL_System.Valve[2].Reset_Cmd := TRUE;
    GVL_System.Valve[3].Reset_Cmd := TRUE;
    GVL_HMI.HMI_ResetAll := FALSE;
END_IF
// MQTT setpoints from FB_MqttManager (parsed from incoming JSON)
GVL_System.Valve[1].MQTT_Setpoint := fbMqttManager.rMqttValveSetpoint[1];
GVL_System.Valve[2].MQTT_Setpoint := fbMqttManager.rMqttValveSetpoint[2];
GVL_System.Valve[3].MQTT_Setpoint := fbMqttManager.rMqttValveSetpoint[3];
GVL_System.bCommandUpdate_MQTT := fbMqttManager.bNewRemoteCommand; 

// MQTT authority is system-wide: HMI_MQTT_bEnable controls the connection,
// and HMI_CommandSource selects whether MQTT commands drive all valves.

// Command source arbitration — choose exactly one source before valve FB calls
CASE GVL_HMI.HMI_CommandSource OF
    E_CommandSource.HMI:
        GVL_System.Valve[1].Active_Setpoint := GVL_System.Valve[1].HMI_Setpoint;
        GVL_System.Valve[2].Active_Setpoint := GVL_System.Valve[2].HMI_Setpoint;
        GVL_System.Valve[3].Active_Setpoint := GVL_System.Valve[3].HMI_Setpoint;
		GVL_System.bCommandUpdate := GVL_System.bCommandUpdate_HMI;
		GVL_HMI.sHMI_mode 		:= TRUE; 
		GVL_HMI.sMannual_mode	:= FALSE;
		GVL_HMI.sMqtt_mode	    := FALSE;     

    E_CommandSource.MQTT:
        IF GVL_HMI.HMI_MQTT_bEnable AND GVL_System.MQTT_Connected THEN
            GVL_System.Valve[1].Active_Setpoint := GVL_System.Valve[1].MQTT_Setpoint;
            GVL_System.Valve[2].Active_Setpoint := GVL_System.Valve[2].MQTT_Setpoint;
            GVL_System.Valve[3].Active_Setpoint := GVL_System.Valve[3].MQTT_Setpoint;
			GVL_System.bCommandUpdate := GVL_System.bCommandUpdate_MQTT;
			GVL_HMI.sMannual_mode	:= FALSE;
			GVL_HMI.sMqtt_mode	    := TRUE;
			GVL_HMI.sHMI_mode 		:= FALSE;   

        END_IF

    E_CommandSource.Manual:
        GVL_System.Valve[1].Active_Setpoint := GVL_System.Valve[1].Manual_Setpoint;
        GVL_System.Valve[2].Active_Setpoint := GVL_System.Valve[2].Manual_Setpoint;
        GVL_System.Valve[3].Active_Setpoint := GVL_System.Valve[3].Manual_Setpoint;
		GVL_System.bCommandUpdate := FALSE;
		GVL_HMI.sMqtt_mode	    := FALSE;
		GVL_HMI.sHMI_mode 		:= FALSE;
		GVL_HMI.sMannual_mode	:= TRUE;  

ELSE
    // Safe fallback for invalid enum values from HMI: keep local HMI authority.
    GVL_System.Valve[1].Active_Setpoint := GVL_System.Valve[1].HMI_Setpoint;
    GVL_System.Valve[2].Active_Setpoint := GVL_System.Valve[2].HMI_Setpoint;
    GVL_System.Valve[3].Active_Setpoint := GVL_System.Valve[3].HMI_Setpoint;
END_CASE

GVL_System.Valve[1].Source := GVL_HMI.HMI_CommandSource;
GVL_System.Valve[2].Source := GVL_HMI.HMI_CommandSource;
GVL_System.Valve[3].Source := GVL_HMI.HMI_CommandSource;


// ============================================================
// STEP 2 — SENSOR I/O
// Reads raw ADC, scales to engineering units, applies LPF.
// Must run before any FB that consumes GVL_System.Sensors.
// ============================================================
fbSensorIO(
    bEnable   := TRUE,
    rLpfAlpha := 0.1,           // 10 % new sample per cycle (moderate filtering)
    stOut     => GVL_System.Sensors
);


// ============================================================
// STEP 3 — VALVE 1
// ============================================================
fbValve1(
    Axis             := Axis_Valve1,
    Active_Setpoint  := GVL_System.Valve[1].Active_Setpoint,
	currentcommandsrc := GVL_HMI.HMI_CommandSource,
 	JogUp            := GVL_IO.bValve1_JogUp_PB,
    JogDown          := GVL_IO.bValve1_JogDown_PB,
    Enable           := TRUE,
    eHomingSelection := MC_DefaultHoming, //MC_Direct,
    Reset            := GVL_System.Valve[1].Reset_Cmd,
    Move_Stop        := GVL_HMI.HMI_Valve1_Stop OR
                       (bManualMode AND GVL_IO.bValve1_JogDown_PB AND
                       NOT GVL_IO.bValve1_JogUp_PB AND GVL_IO.bBottom_position_1),
    ZeroPosition     := GVL_IO.bBottom_position_1,
	TopPosition		 := GVL_IO.bTop_position_1,
  	bUpdate			 := GVL_System.bCommandUpdate,
    bHoming          := GVL_HMI.HMI_Valve1_Homing,
    MoveVelocity     := GVL_Config.VALVE_MOVE_VELOCITY,
    MoveAccel        := GVL_Config.VALVE_MOVE_ACCELERATION,
    MoveDecel        := GVL_Config.VALVE_MOVE_DECELERATION,
    MoveJerk         := GVL_Config.VALVE_MOVE_JERK,
    HomeVelocity     := GVL_Config.VALVE_HOMING_VELOCITY,
    FullStroke_mm    := GVL_Config.VALVE_FULL_STROKE_MM,
    PosTolerance     := GVL_Config.VALVE_POSITION_TOLERANCE,

    Actual_Position  => GVL_System.Valve[1].Actual_Position,
    State            => GVL_System.Valve[1].State,
	currentState_string => GVL_System.Valve[1].currentState_string,
    IsHomed          => GVL_System.Valve[1].IsHomed,
    InPosition       => GVL_System.Valve[1].InPosition,
    IsFault          => GVL_System.Valve[1].IsFault,
    FaultCode        => GVL_System.Valve[1].FaultCode,
    JogUpLed         => GVL_IO.bValve1_JogUp_LED,
    JogDownLed       => GVL_IO.bValve1_JogDown_LED,	
    rTarget_mm       => GVL_HMI.Raw_Valve1_Setpoint,
    rActual_mm       => GVL_HMI.Raw_Valve1_Position,
	lastcommandsrc	 => GVL_System.Valve[1].lastsrc 
);


// ============================================================
// STEP 4 — VALVE 2
// ============================================================
fbValve2(
    Axis             := Axis_Valve2,
    Active_Setpoint  := GVL_System.Valve[2].Active_Setpoint,
	currentcommandsrc := GVL_HMI.HMI_CommandSource,
	JogUp            := GVL_IO.bValve2_JogUp_PB,
    JogDown          := GVL_IO.bValve2_JogDown_PB,
    Enable           := TRUE,
    eHomingSelection := MC_Direct,
    Reset            := GVL_System.Valve[2].Reset_Cmd,
    Move_Stop        := GVL_HMI.HMI_Valve2_Stop OR
                        (bManualMode AND GVL_IO.bValve2_JogDown_PB AND
                         NOT GVL_IO.bValve2_JogUp_PB AND GVL_IO.bBottom_position_2),
    ZeroPosition     := GVL_IO.bBottom_position_2,
    TopPosition      := GVL_IO.bTop_position_2,
	bUpdate			 := GVL_System.bCommandUpdate,
    bHoming          := GVL_HMI.HMI_Valve2_Homing,
    MoveVelocity     := GVL_Config.VALVE_MOVE_VELOCITY,
    MoveAccel        := GVL_Config.VALVE_MOVE_ACCELERATION,
    MoveDecel        := GVL_Config.VALVE_MOVE_DECELERATION,
    MoveJerk         := GVL_Config.VALVE_MOVE_JERK,
    HomeVelocity     := GVL_Config.VALVE_HOMING_VELOCITY,
    FullStroke_mm    := GVL_Config.VALVE_FULL_STROKE_MM,
    PosTolerance     := GVL_Config.VALVE_POSITION_TOLERANCE,

    Actual_Position  => GVL_System.Valve[2].Actual_Position,
    State            => GVL_System.Valve[2].State,
	currentState_string => GVL_System.Valve[2].currentState_string,
    IsHomed          => GVL_System.Valve[2].IsHomed,
    InPosition       => GVL_System.Valve[2].InPosition,
    IsFault          => GVL_System.Valve[2].IsFault,
    FaultCode        => GVL_System.Valve[2].FaultCode,
    JogUpLed         => GVL_IO.bValve2_JogUp_LED,
    JogDownLed       => GVL_IO.bValve2_JogDown_LED,	
    rTarget_mm       => GVL_HMI.Raw_Valve2_Setpoint,
    rActual_mm       => GVL_HMI.Raw_Valve2_Position,
	lastcommandsrc	 => GVL_System.Valve[2].lastsrc
);


// ============================================================
// STEP 5 — VALVE 3
// ============================================================
fbValve3(
    Axis             := Axis_Valve3,
    Active_Setpoint  := GVL_System.Valve[3].Active_Setpoint,
	currentcommandsrc := GVL_HMI.HMI_CommandSource,
	JogUp            := GVL_IO.bValve3_JogUp_PB,
    JogDown          := GVL_IO.bValve3_JogDown_PB,
    Enable           := TRUE,
    eHomingSelection := MC_Direct,
    Reset            := GVL_System.Valve[3].Reset_Cmd,
    Move_Stop        := GVL_HMI.HMI_Valve3_Stop OR
                        (bManualMode AND GVL_IO.bValve3_JogDown_PB AND
                         NOT GVL_IO.bValve3_JogUp_PB AND GVL_IO.bBottom_position_3),
    ZeroPosition     := GVL_IO.bBottom_position_3,
    TopPosition      := GVL_IO.bTop_position_3,
	bUpdate			 := GVL_System.bCommandUpdate,
    bHoming          := GVL_HMI.HMI_Valve3_Homing,
    MoveVelocity     := GVL_Config.VALVE_MOVE_VELOCITY,
    MoveAccel        := GVL_Config.VALVE_MOVE_ACCELERATION,
    MoveDecel        := GVL_Config.VALVE_MOVE_DECELERATION,
    MoveJerk         := GVL_Config.VALVE_MOVE_JERK,
    HomeVelocity     := GVL_Config.VALVE_HOMING_VELOCITY,
    FullStroke_mm    := GVL_Config.VALVE_FULL_STROKE_MM,
    PosTolerance     := GVL_Config.VALVE_POSITION_TOLERANCE,

    Actual_Position  => GVL_System.Valve[3].Actual_Position,
    State            => GVL_System.Valve[3].State,
	currentState_string => GVL_System.Valve[3].currentState_string,
    IsHomed          => GVL_System.Valve[3].IsHomed,
    InPosition       => GVL_System.Valve[3].InPosition,
    IsFault          => GVL_System.Valve[3].IsFault,
    FaultCode        => GVL_System.Valve[3].FaultCode,
	JogUpLed         => GVL_IO.bValve3_JogUp_LED,
    JogDownLed       => GVL_IO.bValve3_JogDown_LED,
    rTarget_mm       => GVL_HMI.Raw_Valve3_Setpoint,
    rActual_mm       => GVL_HMI.Raw_Valve3_Position,
	lastcommandsrc	 => GVL_System.Valve[3].lastsrc
);


// ============================================================
// STEP 6 — AUTO-CLEAR RESET COMMANDS
// Reset is edge-triggered inside FB_ValveControl, so clear here
// to prevent re-trigger on subsequent cycles.
// ============================================================
GVL_System.Valve[1].Reset_Cmd := FALSE;
GVL_HMI.HMI_Valve1_Reset      := FALSE;
GVL_System.Valve[2].Reset_Cmd := FALSE;
GVL_HMI.HMI_Valve2_Reset      := FALSE;
GVL_System.Valve[3].Reset_Cmd := FALSE;
GVL_HMI.HMI_Valve3_Reset      := FALSE;


// ============================================================
// STEP 7 — BUILD TIMESTAMP STRING (YYYY-MM-DD HH:MM:SS)
// Used for MQTT JSON and CSV row timestamps.
// ============================================================
(*fbSysTime(bEnable := TRUE, dwCycle := 1);

sTimestamp := UINT_TO_STRING(fbSysTime.systemTime.wYear);
sTimestamp := CONCAT(sTimestamp, '-');
sTempStr   := UINT_TO_STRING(fbSysTime.systemTime.wMonth);
IF fbSysTime.systemTime.wMonth < 10 THEN sTempStr := CONCAT('0', sTempStr); END_IF
sTimestamp := CONCAT(sTimestamp, sTempStr);
sTimestamp := CONCAT(sTimestamp, '-');
sTempStr   := UINT_TO_STRING(fbSysTime.systemTime.wDay);
IF fbSysTime.systemTime.wDay < 10 THEN sTempStr := CONCAT('0', sTempStr); END_IF
sTimestamp := CONCAT(sTimestamp, sTempStr);
sTimestamp := CONCAT(sTimestamp, ' ');
sTempStr   := UINT_TO_STRING(fbSysTime.systemTime.wHour);
IF fbSysTime.systemTime.wHour < 10 THEN sTempStr := CONCAT('0', sTempStr); END_IF
sTimestamp := CONCAT(sTimestamp, sTempStr);
sTimestamp := CONCAT(sTimestamp, ':');
sTempStr   := UINT_TO_STRING(fbSysTime.systemTime.wMinute);
IF fbSysTime.systemTime.wMinute < 10 THEN sTempStr := CONCAT('0', sTempStr); END_IF
sTimestamp := CONCAT(sTimestamp, sTempStr);
sTimestamp := CONCAT(sTimestamp, ':');
sTempStr   := UINT_TO_STRING(fbSysTime.systemTime.wSecond);
IF fbSysTime.systemTime.wSecond < 10 THEN sTempStr := CONCAT('0', sTempStr); END_IF
sTimestamp := CONCAT(sTimestamp, sTempStr);
*)

// ============================================================
// STEP 8 — MQTT MANAGER
// Populate whole-array buffers (per-element assignment is not
// allowed inside an FB call), then run the manager.
// ============================================================

// Build the array buffers required by FB_MqttManager
aValveSetpoint[1] := GVL_System.Valve[1].Active_Setpoint;
aValveSetpoint[2] := GVL_System.Valve[2].Active_Setpoint;
aValveSetpoint[3] := GVL_System.Valve[3].Active_Setpoint;

aValveActual[1] := GVL_System.Valve[1].Actual_Position;
aValveActual[2] := GVL_System.Valve[2].Actual_Position;
aValveActual[3] := GVL_System.Valve[3].Actual_Position;

aValveSource[1] := GVL_HMI.ACT_Valve1_SourceText;
aValveSource[2] := GVL_HMI.ACT_Valve2_SourceText;
aValveSource[3] := GVL_HMI.ACT_Valve3_SourceText;

fbMqttManager(
    bEnable              := GVL_HMI.HMI_MQTT_bEnable,
    stConfig             := GVL_HMI.HMI_MQTT_Config,
    bApplyConfig         := GVL_HMI.HMI_MQTT_ApplyConfig,
    bPublish             := GVL_HMI.HMI_MQTT_mPublish,
    bEnableStatusPublish := GVL_HMI.HMI_MQTT_Config.bUseStatusPublish,
    tStatusPublishTime   := GVL_HMI.HMI_MQTT_Config.tStatusPublishInterval,
    sStatusTopic         := GVL_HMI.HMI_MQTT_Config.sMainTopic,

    rValveSetpoint       := aValveSetpoint,
    rValveActual         := aValveActual,
    sValveSource         := aValveSource,

    rTemperature_C       := GVL_System.Sensors.rTemperature_C[1],
    rWaterLevel_pct      := GVL_System.Sensors.rWaterLevel_pct,
    rWaterLevel_mm       := GVL_System.Sensors.rWaterLevel_mm,
    sTimestamp           := sTimestamp,

    bConnected           => GVL_System.MQTT_Connected,
    bError               => GVL_System.MQTT_Error,
    nErrorCode           => GVL_System.MQTT_LastErrorCode,
    sErrorMsg            => GVL_System.MQTT_LastErrorMsg,
    sLastRxTopic         => GVL_System.MQTT_LastRxTopic,
    sLastRxPayload       => GVL_System.MQTT_LastRxPayload,
    sJsonStatusPayload   => GVL_System.MQTT_LastJsonStatus,
    bNewRemoteCommand    => GVL_System.MQTT_NewCommand,
	
	LastmsgPub			=> GVL_HMI.ACT_MQTT_LastMsgPubTime,
	LastmsgRcv 			=> GVL_HMI.ACT_MQTT_LastMsgRcvTime,
	currentState_strng		=> GVL_HMI.ACT_MQTT_State
);

// Auto-clear Apply button after one cycle (rising edge consumed inside FB)
GVL_HMI.HMI_MQTT_ApplyConfig := FALSE;


// ============================================================
// STEP 9 — CSV LOGGER
// ============================================================
fbCsvLogger(
    bEnable          := GVL_HMI.HMI_CSV_Enable,
    bForceWrite      := GVL_HMI.WriteTrigger,
    tLogInterval     := GVL_Config.CSV_LOG_INTERVAL_S,
    sBasePath        := GVL_Config.CSV_FILE_PATH,
    sPrefix          := GVL_Config.CSV_FILENAME_PREFIX,
    stValve          := GVL_System.Valve,
    stSensors        := GVL_System.Sensors,

    dtLastWrite      => GVL_System.CSV_LastWriteTime,
    bError           => GVL_System.CSV_FileError,
    sCurrentFilename => GVL_System.CSV_CurrentFile,
    eState           => GVL_System.CSV_LoggerState
);

// Auto-clear write trigger after one cycle
GVL_HMI.WriteTrigger := FALSE;


// ============================================================
// STEP 10 — MIRROR FEEDBACK TO HMI DISPLAY VARIABLES
// All ACT_* variables are read-only from the HMI side.
// ============================================================

// Valve 1 feedback
GVL_HMI.ACT_Valve1_Position  := GVL_System.Valve[1].Actual_Position;
GVL_HMI.ACT_Valve1_State     := GVL_System.Valve[1].currentState_string;
GVL_HMI.ACT_Valve1_Source    := GVL_System.Valve[1].lastsrc;
GVL_HMI.ACT_Valve1_Fault     := GVL_System.Valve[1].IsFault;
GVL_HMI.ACT_Valve1_FaultCode := GVL_System.Valve[1].FaultCode;


// Valve 2 feedback
GVL_HMI.ACT_Valve2_Position  := GVL_System.Valve[2].Actual_Position;
GVL_HMI.ACT_Valve2_State     := GVL_System.Valve[2].currentState_string;
GVL_HMI.ACT_Valve2_Source    := GVL_System.Valve[2].lastsrc;
GVL_HMI.ACT_Valve2_Fault     := GVL_System.Valve[2].IsFault;
GVL_HMI.ACT_Valve2_FaultCode := GVL_System.Valve[2].FaultCode;

// Valve 3 feedback
GVL_HMI.ACT_Valve3_Position  := GVL_System.Valve[3].Actual_Position;
GVL_HMI.ACT_Valve3_State     := GVL_System.Valve[3].currentState_string;
GVL_HMI.ACT_Valve3_Source    := GVL_System.Valve[3].lastsrc;
GVL_HMI.ACT_Valve3_Fault     := GVL_System.Valve[3].IsFault;
GVL_HMI.ACT_Valve3_FaultCode := GVL_System.Valve[3].FaultCode;

// Source text strings (HMI indicators + MQTT JSON sValveSource[])
CASE GVL_System.Valve[1].lastsrc OF
    E_CommandSource.MQTT:   GVL_HMI.ACT_Valve1_SourceText := 'MQTT';
    E_CommandSource.HMI:    GVL_HMI.ACT_Valve1_SourceText := 'HMI';
    E_CommandSource.Manual: GVL_HMI.ACT_Valve1_SourceText := 'Manual';
    ELSE                  GVL_HMI.ACT_Valve1_SourceText := 'NONE';
END_CASE

CASE GVL_System.Valve[2].lastsrc OF
    E_CommandSource.MQTT:   GVL_HMI.ACT_Valve2_SourceText := 'MQTT';
    E_CommandSource.HMI:    GVL_HMI.ACT_Valve2_SourceText := 'HMI';
    E_CommandSource.Manual: GVL_HMI.ACT_Valve2_SourceText := 'Manual';
    ELSE                  GVL_HMI.ACT_Valve2_SourceText := 'NONE';
END_CASE

CASE GVL_System.Valve[3].lastsrc OF
    E_CommandSource.MQTT:   GVL_HMI.ACT_Valve3_SourceText := 'MQTT';
    E_CommandSource.HMI:    GVL_HMI.ACT_Valve3_SourceText := 'HMI';
    E_CommandSource.Manual: GVL_HMI.ACT_Valve3_SourceText := 'Manual';
    ELSE                  GVL_HMI.ACT_Valve3_SourceText := 'NONE';
END_CASE

// Sensor displays
GVL_HMI.ACT_WaterLevel_pct  := GVL_System.Sensors.rWaterLevel_pct;
GVL_HMI.ACT_WaterLevel_mm   := GVL_System.Sensors.rWaterLevel_mm;
GVL_HMI.ACT_Temperature1_C  := GVL_System.Sensors.rTemperature_C[1];
GVL_HMI.ACT_Temperature2_C  := GVL_System.Sensors.rTemperature_C[2];
GVL_HMI.ACT_SensorFault     := GVL_System.Sensors.bAnySensorFault;

// MQTT status
GVL_HMI.ACT_MQTT_Connected   := GVL_System.MQTT_Connected;
GVL_HMI.ACT_MQTT_Error       := GVL_System.MQTT_Error;
GVL_HMI.ACT_MQTT_ErrorMsg    := GVL_System.MQTT_LastErrorMsg;
GVL_HMI.ACT_MQTT_JsonPreview := GVL_System.MQTT_LastJsonStatus;
GVL_HMI.ACT_MQTT_LastRxTopic := GVL_System.MQTT_LastRxTopic;
GVL_HMI.ACT_MQTT_NewCommand  := GVL_System.MQTT_NewCommand;

// CSV status
GVL_HMI.ACT_CSV_CurrentFile   := GVL_System.CSV_CurrentFile;
GVL_HMI.ACT_CSV_LastWriteTime := GVL_System.CSV_LastWriteTime;
GVL_HMI.ACT_CSV_Error         := GVL_System.CSV_FileError;


// ============================================================
// STEP 11 — SYSTEM HEALTH FLAGS
// ============================================================
GVL_System.AnyFaultActive :=
    GVL_System.Valve[1].IsFault OR
    GVL_System.Valve[2].IsFault OR
    GVL_System.Valve[3].IsFault;

GVL_System.AnySensorFault := GVL_System.Sensors.bAnySensorFault;

GVL_System.SystemReady :=
    GVL_System.Valve[1].IsHomed AND
    GVL_System.Valve[2].IsHomed AND
    GVL_System.Valve[3].IsHomed AND
    NOT GVL_System.AnyFaultActive;

GVL_HMI.ACT_SystemReady := GVL_System.SystemReady;

END_PROGRAM

// ---- Functions/FB_SensorIO.TcPOU
(*
============================================================
FUNCTION_BLOCK: FB_SensorIO
============================================================

PURPOSE
  Reads raw analog INT values from GVL_IO (EL3074 / EL3202),
  scales them to engineering units, applies a low-pass filter
  for noise rejection, detects sensor faults, and outputs
  a fully populated ST_SensorData struct.

  Call this block once per PLC cycle in MAIN before any
  other FB that consumes sensor data.

INPUTS
  bEnable         — Master enable; when FALSE outputs hold
                    last valid value and bAnySensorFault = TRUE.
  rLpfAlpha       — Low-pass filter coefficient (0.0–1.0).
                    0.0 = no filtering (pass-through).
                    0.9 = heavy filtering (slow to respond).
                    Default 0.1 gives moderate noise rejection.

OUTPUTS
  stOut           — Fully populated ST_SensorData struct.

WATER LEVEL SCALING
  Linear mapping: (raw − RAW_MIN) / (RAW_MAX − RAW_MIN) × ENG_RANGE
  Scaling constants defined in GVL_Config.

TEMPERATURE SCALING
  EL3202 RTD card outputs tenths of a degree Celsius as INT.
  e.g. raw = 250 → 250 × 0.1 + OFFSET = 25.0 °C

FAULT DETECTION
  Any raw value ≤ GVL_Config.SENSOR_FAULT_THRESHOLD is treated
  as a disconnected or failed sensor (default threshold = -100;
  unconnected GVL_IO stubs initialize to -999).

HARDWARE MAPPING (GVL_IO)
  Water level:   AI_L1V11 (primary), AI_L1V20, AI_L2V21
  Temperature:   AI_Tmp_1, AI_Tmp_2  (EL3202 PT100)
  Position FB:   AI_PosFeedback_1/2/3 (supplementary only)

LIBRARIES
  Tc2_Standard
============================================================
*)

FUNCTION_BLOCK FB_SensorIO
VAR_INPUT
    bEnable     : BOOL := TRUE;     (* Master enable; FALSE holds last value *)
    rLpfAlpha   : REAL := 0.1;      (* Low-pass filter: 0.0=off, 0.9=heavy   *)
END_VAR

VAR_OUTPUT
    stOut       : ST_SensorData;    (* All sensor readings in engineering units *)
END_VAR

VAR
    (* ── Low-pass filter state variables ─────────────────────── *)
    rFilt_WaterLevel    : REAL;
    rFilt_Temp1         : REAL;
    rFilt_Temp2         : REAL;
    rFilt_PosFb         : ARRAY[1..3] OF REAL;

    (* ── Scaled (pre-filter) intermediate values ──────────────── *)
    rRaw_WaterLevel_mm  : REAL;
    rRaw_Temp1_C        : REAL;
    rRaw_Temp2_C        : REAL;
    rRaw_PosFb_mm       : ARRAY[1..3] OF REAL;

    (* ── First-scan flag (initialise filters from first reading) *)
    bFirstScan          : BOOL := TRUE;

    i                   : INT;
END_VAR

// ============================================================
// SECTION 1 — ENABLE GUARD
// ============================================================
IF NOT bEnable THEN
    stOut.bAnySensorFault := TRUE;
    stOut.bWaterLevelFault := TRUE;
    stOut.bTempFault[1]   := TRUE;
    stOut.bTempFault[2]   := TRUE;
    RETURN;
END_IF


// ============================================================
// SECTION 2 — FAULT DETECTION
// A raw value ≤ SENSOR_FAULT_THRESHOLD indicates disconnection.
// ============================================================

stOut.bWaterLevelFault  := GVL_IO.AI_L1V11 <= GVL_Config.SENSOR_FAULT_THRESHOLD;
stOut.bTempFault[1]     := GVL_IO.AI_Tmp_1 <= GVL_Config.SENSOR_FAULT_THRESHOLD;
stOut.bTempFault[2]     := GVL_IO.AI_Tmp_2 <= GVL_Config.SENSOR_FAULT_THRESHOLD;

FOR i := 1 TO 3 DO
    CASE i OF
        1: stOut.bPosFeedbackFault[i] := GVL_IO.AI_PosFeedback_1 <= GVL_Config.SENSOR_FAULT_THRESHOLD;
        2: stOut.bPosFeedbackFault[i] := GVL_IO.AI_PosFeedback_2 <= GVL_Config.SENSOR_FAULT_THRESHOLD;
        3: stOut.bPosFeedbackFault[i] := GVL_IO.AI_PosFeedback_3 <= GVL_Config.SENSOR_FAULT_THRESHOLD;
    END_CASE
END_FOR

stOut.bAnySensorFault :=
    stOut.bWaterLevelFault OR
    stOut.bTempFault[1]    OR
    stOut.bTempFault[2];


// ============================================================
// SECTION 3 — RAW VALUE CAPTURE
// Store raw counts for diagnostics and fault logging.
// ============================================================

stOut.rWaterLevel_raw   := GVL_IO.AI_L1V11;
stOut.rTemperature_raw[1] := GVL_IO.AI_Tmp_1;
stOut.rTemperature_raw[2] := GVL_IO.AI_Tmp_2;
stOut.rPosFeedback_raw[1] := GVL_IO.AI_PosFeedback_1;
stOut.rPosFeedback_raw[2] := GVL_IO.AI_PosFeedback_2;
stOut.rPosFeedback_raw[3] := GVL_IO.AI_PosFeedback_3;


// ============================================================
// SECTION 4 — SCALING TO ENGINEERING UNITS
// Only scale valid readings; keep last valid value on fault.
// ============================================================

IF NOT stOut.bWaterLevelFault THEN
    // Linear: mm = (raw - rawMin) / (rawMax - rawMin) * engRange + engMin
    rRaw_WaterLevel_mm := ScaleLinear(
        INT_TO_REAL(GVL_IO.AI_L1V11),
        INT_TO_REAL(GVL_Config.WATER_LEVEL_RAW_MIN),
        INT_TO_REAL(GVL_Config.WATER_LEVEL_RAW_MAX),
        GVL_Config.WATER_LEVEL_ENG_MIN_MM,
        GVL_Config.WATER_LEVEL_ENG_MAX_MM);
    rRaw_WaterLevel_mm := LIMIT(GVL_Config.WATER_LEVEL_ENG_MIN_MM, rRaw_WaterLevel_mm, GVL_Config.WATER_LEVEL_ENG_MAX_MM);
END_IF

IF NOT stOut.bTempFault[1] THEN
    // EL3202 outputs tenths of a degree: divide by 10 (or apply scale factor)
    rRaw_Temp1_C := INT_TO_REAL(GVL_IO.AI_Tmp_1) * GVL_Config.TEMP_RAW_SCALE_FACTOR + GVL_Config.TEMP_OFFSET_C;
END_IF

IF NOT stOut.bTempFault[2] THEN
    rRaw_Temp2_C := INT_TO_REAL(GVL_IO.AI_Tmp_2) * GVL_Config.TEMP_RAW_SCALE_FACTOR + GVL_Config.TEMP_OFFSET_C;
END_IF

FOR i := 1 TO 3 DO
    IF NOT stOut.bPosFeedbackFault[i] THEN
        CASE i OF
            1: rRaw_PosFb_mm[i] := ScaleLinear(
                    INT_TO_REAL(GVL_IO.AI_PosFeedback_1),
                    INT_TO_REAL(GVL_Config.WATER_LEVEL_RAW_MIN),
                    INT_TO_REAL(GVL_Config.WATER_LEVEL_RAW_MAX),
                    GVL_Config.WATER_LEVEL_ENG_MIN_MM,
                    GVL_Config.VALVE_FULL_STROKE_MM);
            2: rRaw_PosFb_mm[i] := ScaleLinear(
                    INT_TO_REAL(GVL_IO.AI_PosFeedback_2),
                    INT_TO_REAL(GVL_Config.WATER_LEVEL_RAW_MIN),
                    INT_TO_REAL(GVL_Config.WATER_LEVEL_RAW_MAX),
                    GVL_Config.WATER_LEVEL_ENG_MIN_MM,
                    GVL_Config.VALVE_FULL_STROKE_MM);
            3: rRaw_PosFb_mm[i] := ScaleLinear(
                    INT_TO_REAL(GVL_IO.AI_PosFeedback_3),
                    INT_TO_REAL(GVL_Config.WATER_LEVEL_RAW_MIN),
                    INT_TO_REAL(GVL_Config.WATER_LEVEL_RAW_MAX),
                    GVL_Config.WATER_LEVEL_ENG_MIN_MM,
                    GVL_Config.VALVE_FULL_STROKE_MM);
        END_CASE
    END_IF
END_FOR


// ============================================================
// SECTION 5 — LOW-PASS FILTER
// y[n] = alpha * x[n] + (1 - alpha) * y[n-1]
// On first scan, seed the filter with the current reading so
// there is no transient from 0 to actual value.
// ============================================================

IF bFirstScan THEN
    rFilt_WaterLevel := rRaw_WaterLevel_mm;
    rFilt_Temp1      := rRaw_Temp1_C;
    rFilt_Temp2      := rRaw_Temp2_C;
    FOR i := 1 TO 3 DO
        rFilt_PosFb[i] := rRaw_PosFb_mm[i];
    END_FOR
    bFirstScan := FALSE;
ELSE
    rFilt_WaterLevel := rLpfAlpha * rRaw_WaterLevel_mm + (1.0 - rLpfAlpha) * rFilt_WaterLevel;
    rFilt_Temp1      := rLpfAlpha * rRaw_Temp1_C      + (1.0 - rLpfAlpha) * rFilt_Temp1;
    rFilt_Temp2      := rLpfAlpha * rRaw_Temp2_C      + (1.0 - rLpfAlpha) * rFilt_Temp2;
    FOR i := 1 TO 3 DO
        rFilt_PosFb[i] := rLpfAlpha * rRaw_PosFb_mm[i] + (1.0 - rLpfAlpha) * rFilt_PosFb[i];
    END_FOR
END_IF


// ============================================================
// SECTION 6 — WRITE OUTPUTS
// ============================================================

stOut.rWaterLevel_mm   := rFilt_WaterLevel;

// Water level percent: 0–100 based on engineering range
IF GVL_Config.WATER_LEVEL_ENG_MAX_MM > GVL_Config.WATER_LEVEL_ENG_MIN_MM THEN
    stOut.rWaterLevel_pct := LIMIT(0.0,
        (rFilt_WaterLevel - GVL_Config.WATER_LEVEL_ENG_MIN_MM) /
        (GVL_Config.WATER_LEVEL_ENG_MAX_MM - GVL_Config.WATER_LEVEL_ENG_MIN_MM) * 100.0,
        100.0);
ELSE
    stOut.rWaterLevel_pct := 0.0;
END_IF

stOut.rTemperature_C[1] := rFilt_Temp1;
stOut.rTemperature_C[2] := rFilt_Temp2;

FOR i := 1 TO 3 DO
    stOut.rPosFeedback_mm[i] := rFilt_PosFb[i];
END_FOR

(*
============================================================
METHOD: ScaleLinear
============================================================
PURPOSE
  Maps a raw value from [rawMin, rawMax] to [engMin, engMax]
  using linear interpolation.

  result = engMin + (raw - rawMin) / (rawMax - rawMin) * (engMax - engMin)

  If rawMax = rawMin the method returns engMin to avoid
  division by zero.
============================================================
*)
METHOD ScaleLinear : REAL
VAR_INPUT
    rRaw    : REAL;
    rRawMin : REAL;
    rRawMax : REAL;
    rEngMin : REAL;
    rEngMax : REAL;
END_VAR
IF rRawMax = rRawMin THEN
    ScaleLinear := rEngMin;
    RETURN;
END_IF

ScaleLinear := rEngMin + (rRaw - rRawMin) / (rRawMax - rRawMin) * (rEngMax - rEngMin);
END_METHOD

END_FUNCTION_BLOCK

// ---- Functions/FB_ValveControl.TcPOU
(*
============================================================
FUNCTION_BLOCK: FB_ValveControl
============================================================

PURPOSE
  Controls a single irrigation gate valve using TC2_MC2.
  Implements an 8-state PLCopen-compatible state machine
  that manages power, homing, position moves, halts, and
  fault recovery.

STATE MACHINE
  INIT      — Clears all flags, waits for drive ready → HOMING
  HOMING    — Executes MC_Home to find zero reference
  IDLE      — Monitors for setpoint change or homing request
  MOVING    — Executes MC_MoveAbsolute to reach target position
  HOLD      — At target; watches for new setpoint or re-home
  MANNUAL_JOG — Hardware-panel jog mode while Manual source is selected
  HALT      — Stopping via MC_Halt (operator STOP button)
  FAULT     — Latches fault code; waits for Reset command
  RESET     — Executes MC_Reset; then transitions to HOMING

SETPOINT HANDLING
  MAIN selects exactly one command source and passes the resulting
  Active_Setpoint to this FB. This FB only clamps and tracks that
  selected setpoint for motion control.

LIBRARIES
  TC2_MC2
============================================================
*)

FUNCTION_BLOCK FB_ValveControl

VAR_IN_OUT
    Axis                : AXIS_REF;  // Must be linked to an NC axis in I/O mapping
END_VAR

VAR_INPUT
	 // ── Setpoint / source ─────────────────────────────────────
    Active_Setpoint     : REAL;             // Selected target position from MAIN (0.0–100.0 %)
	currentcommandsrc	: E_CommandSource;

    // ── Homing ────────────────────────────────────────────────
    eHomingSelection    : MC_HomingMode;    // Homing mode (MC_Direct sets position without movement)
    bHoming             : BOOL;             // Rising edge: trigger re-home sequence

    // ── Control ───────────────────────────────────────────────
    Enable              : BOOL;             // TRUE = drive powered; FALSE = de-energised
    Reset               : BOOL;             // Rising edge: clear fault and re-home
    Move_Stop           : BOOL;             // TRUE: halt movement immediately
    ZeroPosition        : BOOL;             // Limit switch at home/zero position
	TopPosition			: BOOL;
	bUpdate				: BOOL;
	JogUp               : BOOL;             // Hardware panel jog-up pushbutton
    JogDown             : BOOL;             // Hardware panel jog-down pushbutton

    // ── Motion parameters ─────────────────────────────────────
    // LREAL type required — matches MC_MoveAbsolute VAR_INPUT types exactly.
    // Ref: Beckhoff Infosys → TC2_MC2 → MC_MoveAbsolute
    MoveVelocity        : LREAL;    // mm/s    — normal travel speed
    MoveAccel           : LREAL;    // mm/s²   — acceleration ramp
    MoveDecel           : LREAL;    // mm/s²   — deceleration ramp
    MoveJerk            : LREAL;    // mm/s³   — jerk limit; 0.0 = trapezoidal profile
    HomeVelocity        : LREAL;    // mm/s    — reference; actual speed set in NC Homing tab

    // ── Scaling ───────────────────────────────────────────────
    FullStroke_mm       : REAL;     // mm — axis travel at 100 % open (calibrate to hardware)
    PosTolerance        : REAL;     // %  — in-position dead-band
END_VAR

VAR_OUTPUT
    // ── Position feedback ─────────────────────────────────────
    Actual_Position     : REAL;             // Current valve opening (0.0–100.0 %)
    InPosition          : BOOL;             // TRUE when |actual - setpoint| <= PosTolerance
    rActual_mm          : LREAL;            // Raw axis position in mm
    rTarget_mm          : LREAL := 0.0;     // Active target in mm
	lastcommandsrc		: E_CommandSource;

    // ── State ─────────────────────────────────────────────────
    State               : E_ValveState;     // Current state machine state (for HMI display)
	currentState_string : STRING;

    // ── Status flags ──────────────────────────────────────────
    IsHomed             : BOOL;             // TRUE once homing completed successfully
    IsMoving            : BOOL;             // TRUE while axis is physically moving
    IsFault             : BOOL;             // TRUE while in FAULT state
    FaultCode           : UDINT;            // MC2 ErrorID — see Beckhoff error code list
	JogUpLed            : BOOL;             // Hardware panel up LED (blink while jogging, solid at top limit)
    JogDownLed          : BOOL;             // Hardware panel down LED (blink while jogging, solid at bottom limit)
END_VAR

VAR
    // ── TC2_MC2 function block instances ──────────────────────
    // Declared at FB level so they retain state between PLC cycles.
    // Ref: Beckhoff Infosys → TC2_MC2 → General Information
    fbPower             : MC_Power;
    fbHome              : MC_Home;
    fbMoveAbs           : MC_MoveAbsolute;
    fbReadPos           : MC_ReadActualPosition;
    fbHalt              : MC_Halt;
    fbReset_MC          : MC_Reset;
	fbSetPos			: MC_SetPosition;
	fbJog		        : MC_Jog;
	

    // ── State machine ─────────────────────────────────────────
    eState              : E_ValveState := E_ValveState.INIT;

    // ── Selected setpoint tracking ────────────────────────────
    rActiveSetpoint     : REAL  := 0.0;
    rPrev_Active_SP     : REAL  := -999.0;  // -999 ensures first selected value is always applied

    // ── PLCopen Execute flags ─────────────────────────────────
    // Set TRUE on state entry → MC FB receives rising edge.
    // Set FALSE on Done/Error → FB resets, ready for next trigger.
    // Ref: PLCopen Motion Control Part 1, Section 4
    bExecHome           : BOOL;
    bExecMove           : BOOL;
    bExecReset          : BOOL;
    bExecHalt           : BOOL;
	bExecJogMove        : BOOL;

    // ── Edge detection ────────────────────────────────────────
    rtReset             : R_TRIG;
    rtZeroPosition      : R_TRIG; //not used
    rtHoming            : R_TRIG;
	rtUpdate			: R_TRIG;

    // ── Internal working variables ────────────────────────────
    bAxisReady          : BOOL;
    bManualMode         : BOOL;
    bJogUpAllowed       : BOOL;
    bJogDownAllowed     : BOOL;
	bJogUpActive        : BOOL;
    bJogDownActive      : BOOL;
    bBlink              : BOOL;
	fbJogBlinkTimer     : TON;
    nBlinkCounter       : UDINT;
    MoveDone            : BOOL;
    tempSetpoint        : REAL;
END_VAR

// ============================================================
// SECTION 1 — EDGE DETECTION
// R_TRIG output Q is TRUE for exactly one PLC cycle on a
// rising edge. Ensures button presses trigger exactly once.
// ============================================================
rtReset(CLK := Reset);
rtHoming(CLK := bHoming);
rtUpdate(CLK := bUpdate);


bManualMode := (currentcommandsrc = E_CommandSource.Manual);
bJogUpAllowed := bManualMode AND JogUp AND NOT JogDown AND NOT TopPosition AND NOT IsFault;
bJogDownAllowed := bManualMode AND JogDown AND NOT JogUp AND NOT ZeroPosition AND NOT IsFault;


// ReadStatus must be called every cycle to keep Axis state current
Axis.ReadStatus();


// ============================================================
// SECTION 2 — SELECTED SETPOINT TRACKING
// MAIN performs command-source arbitration before this FB is called.
// This FB accepts only the already selected setpoint, clamps it, and
// updates the motion target when that selected value changes. Manual
// jog inputs override the selected setpoint only while Manual source
// is active; simultaneous JogUp/JogDown input is ignored.
// ============================================================

IF rtUpdate.Q  THEN  //Active_Setpoint <> rPrev_Active_SP
    rActiveSetpoint := LIMIT(0.0, Active_Setpoint, 100.0);
    rPrev_Active_SP := Active_Setpoint;
END_IF

// Convert percentage setpoint to axis units (mm)
rTarget_mm := REAL_TO_LREAL(rActiveSetpoint / 100.0 * FullStroke_mm);


// ============================================================
// SECTION 3 — MC_Power
// Enable drive power. Disable during FAULT to allow safe state.
// Catches unexpected drive errors from any running state.
// ============================================================
fbPower(
    Axis            := Axis,
    Enable          := Enable AND (eState <> E_ValveState.FAULT),
    Enable_Positive := TRUE AND NOT TopPosition,    // NC software limits protect max travel
    Enable_Negative := TRUE,    // NC software limits protect min travel
    Override        := 100.0    // 100 % velocity override = full programmed speed
);
bAxisReady := fbPower.Status AND NOT fbPower.Error;

// Trap unexpected drive fault from any non-fault/non-reset state
IF fbPower.Error AND
   eState <> E_ValveState.FAULT AND
   eState <> E_ValveState.RESET AND
   eState <> E_ValveState.INIT
THEN
    FaultCode := fbPower.ErrorID;
    eState    := E_ValveState.FAULT;
END_IF


// ============================================================
// SECTION 4 — MC_ReadActualPosition
// Read current axis position every cycle.
// rActual_mm is then converted to a percentage.
// ============================================================
(*
IF TopPosition THEN
	fbSetPos (
		Axis := Axis,
		Execute := TRUE,
		Position := FullStroke_mm
		//Mode
		);	
	IF fbSetPos.Done THEN
		fbSetPos (Execute := FALSE, Axis := Axis);
		rActiveSetpoint := Actual_Position;  // Adopt current position as new setpoint
		rPrev_Active_SP := Active_Setpoint;   // Hold until selected setpoint changes
	END_IF
END_IF 
*)
fbReadPos(
    Axis   := Axis,
    Enable := fbPower.Status
);
IF fbReadPos.Valid THEN
    rActual_mm := fbReadPos.Position;
END_IF

// Convert mm to percentage of full stroke
IF FullStroke_mm > 0.0 THEN
    Actual_Position := LREAL_TO_REAL(rActual_mm / REAL_TO_LREAL(FullStroke_mm)) * 100.0;
    Actual_Position := LIMIT(0.0, Actual_Position, 100.0);
ELSE
    Actual_Position := 0.0;  // Guard: division by zero if FullStroke_mm not configured
END_IF

// In-position flag: TRUE when within tolerance of active setpoint
InPosition := ABS(Actual_Position - rActiveSetpoint) <= PosTolerance;


// Manual source forces the valve into hardware-panel jog mode from normal states.
// FAULT and RESET remain latched/safe; INIT waits for drive power first.
IF bManualMode AND
   eState <> E_ValveState.MANNUAL_JOG AND
   eState <> E_ValveState.FAULT AND
   eState <> E_ValveState.RESET AND
   eState <> E_ValveState.INIT
THEN
    bExecHome := FALSE;
    bExecMove := FALSE;
    bExecJogMove := FALSE;
    fbHome(Axis := Axis, Execute := FALSE);
    fbMoveAbs(Axis := Axis, Execute := FALSE);
    eState := E_ValveState.MANNUAL_JOG;
END_IF



// ============================================================
// SECTION 5 — STATE MACHINE
// Each state is responsible for:
//   a) Setting/clearing Execute flags for MC FBs
//   b) Monitoring completion/error conditions
//   c) Transitioning to the next state
// ============================================================
CASE eState OF

    // ----------------------------------------------------------
    // INIT: Clear all Execute flags; wait for drive ready.
    // Drive ready = MC_Power.Status = TRUE, no error.
    // ----------------------------------------------------------
    E_ValveState.INIT:
		currentState_string := 'INIT';
        bExecHome  := FALSE;
        bExecMove  := FALSE;
        bExecReset := FALSE;
        bExecHalt  := FALSE;
		bExecJogMove := FALSE;

        IF bAxisReady THEN
            IF bManualMode THEN
                eState := E_ValveState.MANNUAL_JOG;
            ELSE
                eState := E_ValveState.HOMING;
            END_IF
        END_IF

    // ----------------------------------------------------------
    // HOMING: Execute MC_Home to establish zero reference.
    // Position = 0.0 mm means valve fully closed.
    // ZeroPosition (limit switch) is the calibration cam signal.
    // ----------------------------------------------------------
    E_ValveState.HOMING:
		currentState_string := 'HOMING';
        bExecHome := TRUE;

        fbHome(
            Axis            := Axis,
            Execute         := bExecHome,
            Position        := 0.0,             // Home = 0 mm = fully closed
            HomingMode      := eHomingSelection, // MC_Direct sets position without movement
            bCalibrationCam := ZeroPosition      // Wired to limit switch in GVL_IO
        );
		
		        // Operator STOP button: halt cleanly
        IF Move_Stop THEN
            bExecHalt := TRUE;
            eState    := E_ValveState.HALT;
        END_IF

        IF fbHome.Done THEN
            bExecHome := FALSE;
            fbHome(Axis := Axis, Execute := bExecHome);  // Clear Execute cleanly
            IsHomed   := TRUE;
			rActiveSetpoint := 0;       // Adopt home position as new setpoint
			rPrev_Active_SP := -999.0; // Reapply selected setpoint on next scan
            eState    := E_ValveState.IDLE;
        ELSIF fbHome.Error THEN
            bExecHome := FALSE;
            fbHome(Axis := Axis, Execute := bExecHome);  // Clear Execute cleanly
            FaultCode := fbHome.ErrorID;
            eState    := E_ValveState.FAULT;
        END_IF

    // ----------------------------------------------------------
    // IDLE: Monitoring for a new setpoint or re-home request.
    // Transition to MOVING only after successful homing.
    // ----------------------------------------------------------
    E_ValveState.IDLE:
		currentState_string := 'IDLE';
        bExecMove := FALSE;

        IF rtHoming.Q THEN
            IsHomed := FALSE;
            eState  := E_ValveState.HOMING;
        END_IF

 		IF IsHomed AND ABS(rActiveSetpoint - Actual_Position) > PosTolerance THEN
            bExecMove := TRUE;
            eState    := E_ValveState.MOVING;
        END_IF

    // ----------------------------------------------------------
    // MOVING: Execute MC_MoveAbsolute to reach target position.
    // Transitions:
    //   Done          → HOLD (at position)
    //   CommandAborted→ IDLE (setpoint changed during move)
    //   Error         → FAULT
    //   Move_Stop     → HALT (operator emergency stop)
    // ----------------------------------------------------------
    E_ValveState.MOVING:
		currentState_string := 'MOVING_ABS';
        fbMoveAbs(
            Axis         := Axis,
            Execute      := bExecMove,
            Position     := rTarget_mm,
            Velocity     := MoveVelocity,
            Acceleration := MoveAccel,
            Deceleration := MoveDecel,
            Jerk         := MoveJerk,     // 0.0 = trapezoidal; >0 = S-curve
            BufferMode   := MC_BlendingNext,
            Active       => IsMoving,
            Done         => MoveDone
        );
		lastcommandsrc := currentcommandsrc;
        // Operator STOP button: halt cleanly
        IF Move_Stop THEN
            bExecHalt := TRUE;
            eState    := E_ValveState.HALT;
        END_IF

        IF fbMoveAbs.Done THEN
            bExecMove := FALSE;
            fbMoveAbs(Axis := Axis, Execute := bExecMove);  // Clear Execute cleanly
            
			eState    := E_ValveState.HOLD;
        ELSIF fbMoveAbs.CommandAborted THEN
            bExecMove := FALSE;
            fbMoveAbs(Axis := Axis, Execute := bExecMove);  // Clear Execute cleanly
            eState    := E_ValveState.IDLE;  // Re-evaluate setpoint on next cycle
        ELSIF fbMoveAbs.Error THEN
            bExecMove := FALSE;
            fbMoveAbs(Axis := Axis, Execute := bExecMove);  // Clear Execute cleanly
            FaultCode := fbMoveAbs.ErrorID;
            eState    := E_ValveState.FAULT;
        END_IF

    // ----------------------------------------------------------
    // HOLD: Valve is at target position.
    // Monitors for new setpoint (→ MOVING) or re-home (→ HOMING).
    // ----------------------------------------------------------
    E_ValveState.HOLD:
	currentState_string := 'HOLD';
        IsMoving  := FALSE;
        bExecMove := FALSE;

        IF ABS(rActiveSetpoint - Actual_Position) > PosTolerance THEN
            bExecMove := TRUE;
            eState    := E_ValveState.MOVING;
        END_IF

        IF rtHoming.Q THEN
            IsHomed := FALSE;
            eState  := E_ValveState.HOMING;
        END_IF

    // ----------------------------------------------------------
    // MANNUAL_JOG: Hardware-panel jog mode selected by system source.
    // Up/down pushbuttons move toward travel limits while held.
    // Bottom limit is NOT tied to MC_Power negative enable because it is the homing cam.
    // ----------------------------------------------------------
    E_ValveState.MANNUAL_JOG:
	currentState_string := 'MANNUAL_JOG';
	
	    // Cancel normal absolute motion while in manual jog mode
    bExecMove := FALSE;
    bExecHome := FALSE;
    bExecReset := FALSE;

    fbMoveAbs(Axis := Axis, Execute := FALSE);
    fbHome(Axis := Axis, Execute := FALSE);
	
	fbJog (
		Axis 			:= Axis,
		JogForward 		:= bJogUpAllowed,
		JogBackwards	:= bJogDownAllowed,
		Mode			:= E_JogMode.MC_JOGMODE_STANDARD_SLOW,
		Active			=> IsMoving
	);
	IF IsMoving THEN
	lastcommandsrc := currentcommandsrc;
	END_IF
	bJogDownActive := IsMoving AND bJogDownAllowed;
	bJogUpActive   := IsMoving AND bJogUpAllowed;
	
        // If the axis was jogging, stop it cleanly
     IF IsMoving AND NOT bJogDownAllowed AND NOT bJogUpAllowed THEN
		 //bJogWasActive := FALSE;
            bExecHalt := TRUE;
            eState := E_ValveState.HALT;
        ELSE
            //IsMoving := FALSE;
        END_IF

    // Jog motion error handling
    IF fbJog.Error THEN
        //bJogWasActive := FALSE;
        FaultCode := fbJog.ErrorID;
        eState := E_ValveState.FAULT;
    END_IF

    // STOP button while jogging
    IF Move_Stop THEN
       // bJogWasActive := FALSE;
        bExecHalt := TRUE;
        eState := E_ValveState.HALT;
    END_IF

    // Leave manual jog mode when command source changes
    IF NOT bManualMode THEN
       // bJogWasActive := FALSE;
        // Adopt current position as the new target
        rActiveSetpoint := Actual_Position;
        rPrev_Active_SP := Active_Setpoint;

        eState := E_ValveState.IDLE;
    END_IF
			

    // ----------------------------------------------------------
    // FAULT: Drive or motion error detected.
    // Latches IsFault = TRUE; waits for Reset command.
    // ──────────────────────────────────────────────────────────
    E_ValveState.FAULT:
	currentState_string := 'FAULT';
        IsFault   := TRUE;
        IsMoving  := FALSE;
        bExecHome := FALSE;
        bExecMove := FALSE;
		bExecJogMove := FALSE;

        IF rtReset.Q THEN
            bExecReset := TRUE;
            eState     := E_ValveState.RESET;
        END_IF

    // ----------------------------------------------------------
    // HALT: MC_Halt stops the axis gracefully.
    // After halt: stay at current position (update setpoint).
    // Reset button returns to IDLE.
    // ----------------------------------------------------------
    E_ValveState.HALT:
	currentState_string := 'HALT';
        fbHalt(
            Axis         := Axis,
            Execute      := bExecHalt,
            Deceleration := MoveDecel,
            Jerk         := MoveJerk,
            BufferMode   := MC_Aborting
        );

        IF fbHalt.Done THEN
            bExecHalt       := FALSE;
            fbHalt(Axis := Axis, Execute := bExecHalt);  // Clear Execute cleanly
            rActiveSetpoint := Actual_Position;  // Adopt current position as new setpoint
            rPrev_Active_SP := Active_Setpoint;   // Hold until selected setpoint changes
			
			// After stopping from manual jog, return to manual jog mode
			IF bManualMode THEN
				eState := E_ValveState.MANNUAL_JOG;
			ELSIF rtReset.Q THEN
				eState := E_ValveState.IDLE;
			END_IF
			
        ELSIF fbHalt.Error THEN
            bExecHalt := FALSE;
            fbHalt(Axis := Axis, Execute := bExecHalt);  // Clear Execute cleanly
            FaultCode := fbHalt.ErrorID;
            eState    := E_ValveState.FAULT;
        END_IF
		
		IF rtReset.Q THEN
			IF bManualMode THEN
				eState := E_ValveState.MANNUAL_JOG;
			ELSE
				eState := E_ValveState.IDLE;
			END_IF
		END_IF
    // ----------------------------------------------------------
    // RESET: Clear drive error with MC_Reset, then re-home.
    // IsHomed is cleared because stepper may have lost position.
    // ----------------------------------------------------------
    E_ValveState.RESET:
	currentState_string := 'RESET';
        fbReset_MC(
            Axis    := Axis,
            Execute := bExecReset
        );

        IF fbReset_MC.Done THEN
            bExecReset := FALSE;
            IsFault    := FALSE;
            FaultCode  := 0;
            IsHomed    := FALSE;  // Must re-home after drive reset
            eState     := E_ValveState.HOMING;
        ELSIF fbReset_MC.Error THEN
            bExecReset := FALSE;  // Next Reset press will retry
            FaultCode  := fbReset_MC.ErrorID;
            // Stay in RESET
        END_IF

ELSE
    // Unknown state — safety fallback: restart from INIT
    eState := E_ValveState.INIT;

END_CASE



IF eState <> E_ValveState.MANNUAL_JOG THEN
    bJogUpActive := FALSE;
    bJogDownActive := FALSE;
END_IF

// ============================================================
// SECTION 5.5 — MANUAL JOG LED LOGIC
// Blink while jogging.
// Solid ON when corresponding limit switch is reached.
// ============================================================

fbJogBlinkTimer(
    IN := (eState = E_ValveState.MANNUAL_JOG)
          AND (bJogUpActive OR bJogDownActive)
          AND NOT fbJogBlinkTimer.Q,
    PT := T#1MS
);

IF fbJogBlinkTimer.Q THEN
    bBlink := NOT bBlink;
END_IF

// UP / OPEN LED
// Blinks while jogging up.
// Solid ON when top/open limit is reached.
JogUpLed :=
    TopPosition OR
    (
        (eState = E_ValveState.MANNUAL_JOG)
        AND bJogUpActive
        AND bBlink
    );

// DOWN / CLOSE LED
// Blinks while jogging down.
// Solid ON when zero/closed limit is reached.
JogDownLed :=
    ZeroPosition OR
    (
        (eState = E_ValveState.MANNUAL_JOG)
        AND bJogDownActive
        AND bBlink
    );


// ============================================================
// SECTION 6 — OUTPUT ASSIGNMENT
// Mirror internal state to VAR_OUTPUT for MAIN and HMI.
// ============================================================
State   := eState;
IsFault := (eState = E_ValveState.FAULT);

END_FUNCTION_BLOCK

// ---- Functions/FB_CSVLogger.TcPOU
(*
============================================================
FUNCTION_BLOCK: FB_CsvLogger
============================================================

PURPOSE
  Appends one CSV row per log interval to a monthly log file
  on the IPC local filesystem (C:\TwinCAT\3.1\Boot\Log\).

FILE NAMING
  <sBasePath><sPrefix><YYYY-MM>.csv
  Example: C:\TwinCAT\3.1\Boot\Log\IrrigationLog_2026-04.csv

CSV COLUMNS
  Timestamp, V1_Setpoint_%, V1_Actual_%, V1_Source, V1_State,
  V2_Setpoint_%, V2_Actual_%, V2_Source, V2_State,
  V3_Setpoint_%, V3_Actual_%, V3_Source, V3_State,
  WaterLevel_mm, WaterLevel_%, Temperature1_C, Temperature2_C

STATE MACHINE
  CSV_IDLE       — Waiting for trigger (timer or force write)
  CSV_PREPARE    — Build filename, check if file exists
  CSV_OPEN       — Open file in append mode
  CSV_WRITE_HDR  — Write column header (new file only)
  CSV_WRITE_ROW  — Append one data row
  CSV_CLOSE      — Close file handle
  CSV_ERROR      — I/O error; waits for next trigger to retry

NOTES
  - File I/O FBs are non-blocking; each step may span PLC cycles.
  - bForceWrite forces a row write outside the normal interval.
  - Header is written only on the first write to a new file.

LIBRARIES
  Tc2_Utilities (FB_FileOpen, FB_FileWrite, FB_FileClose, FB_EnumFindFileEntry)
  Tc2_System    (FB_LocalSystemTime)
============================================================
*)

FUNCTION_BLOCK FB_CsvLogger

VAR_INPUT
    bEnable         : BOOL := TRUE;         (* Master enable; FALSE skips all logging    *)
    bForceWrite     : BOOL;                 (* Rising edge: write a row immediately      *)
    tLogInterval    : TIME;                 (* Periodic write interval (e.g. T#15M)      *)
    sBasePath       : STRING(128);          (* Folder path including trailing backslash  *)
    sPrefix         : T_MaxString;          (* Filename prefix (e.g. 'IrrigationLog_')   *)
    stValve         : ARRAY[1..3] OF ST_ValveData;  (* Valve runtime data from GVL_System *)
    stSensors       : ST_SensorData;        (* Sensor readings from FB_SensorIO          *)
END_VAR

VAR_OUTPUT
    bBusy           : BOOL;                 (* TRUE while file I/O is in progress        *)
    bError          : BOOL;                 (* TRUE on file I/O error                    *)
    nErrorCode      : UDINT;               (* Error code from file FB (0 = OK)           *)
    dtLastWrite     : DT;                   (* Timestamp of last successful row write     *)
    sCurrentFilename : STRING(128);         (* Active filename (without path)             *)
    sCurrentFile    : STRING(128);          (* Full file path currently being written     *)
    eState          : E_CSVLogState := E_CSVLogState.CSV_IDLE;
END_VAR

VAR
    (* File I/O FBs *)
    fbFileOpen      : FB_FileOpen;
    fbFileWrite     : FB_FileWrite;
    fbFileClose     : FB_FileClose;
    hFilenumber     : UINT;
    cbLen           : UDINT;

    (* Timing *)
    tIntervalTimer  : TON;
    bForceEdge      : R_TRIG;
    bTriggerWrite   : BOOL;

    (* Date/time *)
    fbGetTime       : FB_LocalSystemTime;
    sTimestamp      : STRING(24);   (* YYYY-MM-DD HH:MM:SS *)
    nYear           : UINT;
    nMonth          : UINT;
    sYear           : STRING(8);
    sMonth          : STRING(4);

    (* File existence check *)
    fbEnum          : FB_EnumFindFileEntry;
    bEnumStart      : BOOL;
    bFileExists     : BOOL;

    (* String building *)
    sLine           : STRING(512);
    sHeader         : STRING(512);
    sSource         : STRING(8);    (* Temp variable for source text per valve *)
END_VAR

(* ============================================================
   GET CURRENT TIME every PLC cycle.
   fbGetTime.systemTime holds year, month, day, hour, min, sec.
   ============================================================ *)
fbGetTime(bEnable := TRUE, dwCycle := 1);


(* ============================================================
   ENABLE GUARD
   When disabled, reset timers but stay in IDLE.
   ============================================================ *)
IF NOT bEnable THEN
    tIntervalTimer(IN := FALSE);
    eState := E_CSVLogState.CSV_IDLE;
    RETURN;
END_IF


(* ============================================================
   TRIGGER LOGIC
   bTriggerWrite fires on:
     a) interval timer expiry (tLogInterval)
     b) rising edge on bForceWrite (manual button)
   ============================================================ *)
bForceEdge(CLK := bForceWrite);
tIntervalTimer(IN := TRUE, PT := tLogInterval);
bTriggerWrite := tIntervalTimer.Q OR bForceEdge.Q;

IF tIntervalTimer.Q THEN
    tIntervalTimer(IN := FALSE);   (* Reset timer for next interval *)
END_IF


(* ============================================================
   STATE MACHINE
   ============================================================ *)
CASE eState OF

    (* ----------------------------------------------------------
       CSV_IDLE — waiting for write trigger
       ---------------------------------------------------------- *)
    E_CSVLogState.CSV_IDLE:
        bBusy := FALSE;

        IF bTriggerWrite THEN
            bFileExists := FALSE;
            bEnumStart  := TRUE;
            eState      := E_CSVLogState.CSV_PREPARE;
        END_IF

    (* ----------------------------------------------------------
       CSV_PREPARE — build filename, check if file already exists.
       Monthly rotation: IrrigationLog_YYYY-MM.csv
       ---------------------------------------------------------- *)
    E_CSVLogState.CSV_PREPARE:
        bBusy := TRUE;

        nYear  := fbGetTime.systemTime.wYear;
        nMonth := fbGetTime.systemTime.wMonth;
        sYear  := UINT_TO_STRING(nYear);
        sMonth := UINT_TO_STRING(nMonth);

        IF nMonth < 10 THEN
            sMonth := CONCAT('0', sMonth);   (* Zero-pad single-digit month *)
        END_IF

        sCurrentFilename := CONCAT(sPrefix, sYear);
        sCurrentFilename := CONCAT(sCurrentFilename, '-');
        sCurrentFilename := CONCAT(sCurrentFilename, sMonth);
        sCurrentFilename := CONCAT(sCurrentFilename, '.csv');
        sCurrentFile     := CONCAT(sBasePath, sCurrentFilename);

        (* Use FB_EnumFindFileEntry to check if file already exists.
           If it does, we skip the header row. *)
        IF bEnumStart THEN
            fbEnum(
                sPathName := sCurrentFile,
                eCmd      := eEnumCmd_First,
                bExecute  := TRUE,
                tTimeout  := T#5S);
            bEnumStart := FALSE;
        ELSE
            fbEnum(
                sPathName := sCurrentFile,
                eCmd      := eEnumCmd_Next,
                bExecute  := FALSE,
                tTimeout  := T#5S);
        END_IF

        IF NOT fbEnum.bBusy THEN
            fbEnum(bExecute := FALSE);
            IF fbEnum.bError THEN
                bFileExists := FALSE;   (* Error means file not found = new file *)
            ELSE
                bFileExists := (fbEnum.stFindFile.sFileName <> '');
            END_IF
            eState := E_CSVLogState.CSV_OPEN;
        END_IF

    (* ----------------------------------------------------------
       CSV_OPEN — open file in append mode (creates if not exists)
       ---------------------------------------------------------- *)
    E_CSVLogState.CSV_OPEN:
        fbFileOpen(
            sPathName := sCurrentFile,
            nMode     := FOPEN_MODEAPPEND,
            bExecute  := TRUE,
            hFile     => hFilenumber);

